SPLINE
SPL {X  -160.284, Y  +717.322, Z    +0.000, E1   -73.988, E3 +103602.756}
SPL {X  -157.512, Y  +726.783, Z    +0.000, E1   -73.653, E3 +103611.470}
SPL {X  -155.383, Y  +732.911, Z    +0.000, E1   -73.297, E3 +103618.397}
SPL {X  -152.193, Y  +740.900, Z    +0.000, E1   -73.135, E3 +103624.475}
SPL {X  -148.880, Y  +748.126, Z    +0.000, E1   -72.716, E3 +103632.256}
SPL {X  -144.434, Y  +756.610, Z    +0.000, E1   -72.338, E3 +103640.106}
SPL {X  -141.532, Y  +761.573, Z    +0.000, E1   -71.800, E3 +103646.746}
SPL {X  -138.580, Y  +766.249, Z    +0.000, E1   -71.449, E3 +103651.808}
SPL {X  -134.851, Y  +771.704, Z    +0.000, E1   -71.081, E3 +103657.203}
SPL {X  -130.513, Y  +777.511, Z    +0.000, E1   -70.561, E3 +103663.386}
SPL {X  -127.002, Y  +781.850, Z    +0.000, E1   -69.819, E3 +103669.241}
SPL {X  -118.977, Y  +790.758, Z    +0.000, E1   -71.976, E3 +103665.358}
SPL {X   -54.135, Y  +832.054, Z    +0.000, E1   -56.519, E3 +103841.284}
ENDSPLINE

SPLINE
SPL {X  -119.915, Y  +789.781, Z    +0.000, E1   -62.637, E3 +104008.899}
SPL {X  -140.675, Y  +762.967, Z    +0.000, E1   -56.489, E3 +104009.241}
SPL {X  -155.138, Y  +733.569, Z    +0.000, E1   -46.550, E3 +104011.546}
SPL {X  -162.699, Y  +706.626, Z    +0.000, E1   -30.890, E3 +104010.587}
SPL {X  -165.420, Y  +684.230, Z    +0.000, E1   -11.665, E3 +104010.338}
SPL {X  -165.650, Y  +673.379, Z    +0.000, E1    +0.036, E3 +104008.998}
SPL {X  -165.650, Y  +670.223, Z    +0.000, E1    +7.575, E3 +104008.439}
SPL {X  -165.650, Y  +666.568, Z    +0.000, E1   +16.799, E3 +104008.416}
SPL {X  -165.650, Y  +661.246, Z    +0.000, E1   +30.569, E3 +104008.196}
SPL {X  -165.650, Y  +652.403, Z    +0.000, E1   +48.665, E3 +104007.834}
SPL {X  -165.650, Y  +637.100, Z    +0.000, E1   +69.106, E3 +104004.174}
SPL {X  -165.650, Y  +616.344, Z    +0.000, E1   +74.941, E3 +104007.424}
SPL {X  -165.650, Y  +575.817, Z    +0.000, E1   +77.800, E3 +104016.353}
SPL {X  -161.405, Y  +341.238, Z    +0.000, E1   +76.606, E3 +104107.653}
SPL {X  -146.302, Y  +300.811, Z    +0.000, E1   +78.008, E3 +104108.770}
ENDSPLINE

SPLINE
SPL {X  -147.825, Y  +303.750, Z    +0.000, E1   +76.548, E3 +104123.202}
SPL {X  -148.167, Y  +304.430, Z    +0.000, E1   +75.276, E3 +104135.295}
ENDSPLINE

SPLINE
SPL {X  -146.983, Y  +302.107, Z    +0.000, E1   +74.473, E3 +104143.775}
SPL {X  -146.624, Y  +301.420, Z    +0.000, E1   +73.294, E3 +104154.259}
SPL {X  -144.830, Y  +298.101, Z    +0.000, E1   +72.333, E3 +104163.783}
SPL {X  -140.483, Y  +290.724, Z    +0.000, E1   +71.922, E3 +104170.940}
SPL {X  -135.200, Y  +282.788, Z    +0.000, E1   +71.482, E3 +104178.285}
SPL {X  -130.835, Y  +276.902, Z    +0.000, E1   +70.642, E3 +104186.187}
SPL {X  -127.149, Y  +272.325, Z    +0.000, E1   +70.073, E3 +104191.439}
SPL {X  -123.924, Y  +268.578, Z    +0.000, E1   +70.633, E3 +104191.255}
SPL {X  -115.163, Y  +259.431, Z    +0.000, E1   +74.058, E3 +104182.365}
SPL {X   -55.479, Y  +222.417, Z    +0.000, E1   +56.403, E3 +104368.218}
ENDSPLINE

SPLINE
SPL {X  -130.757, Y  +276.802, Z    +0.000, E1   +58.343, E3 +104524.155}
SPL {X  -154.788, Y  +319.502, Z    +0.000, E1   +45.389, E3 +104528.353}
SPL {X  -161.887, Y  +343.393, Z    +0.000, E1   +32.461, E3 +104528.809}
SPL {X  -164.949, Y  +363.277, Z    +0.000, E1   +17.059, E3 +104528.084}
SPL {X  -165.591, Y  +374.070, Z    +0.000, E1    +6.781, E3 +104527.747}
SPL {X  -165.650, Y  +380.752, Z    +0.000, E1    -0.182, E3 +104526.743}
SPL {X  -165.650, Y  +385.053, Z    +0.000, E1   -10.073, E3 +104526.210}
SPL {X  -165.650, Y  +388.847, Z    +0.000, E1   -19.524, E3 +104526.175}
SPL {X  -165.650, Y  +394.451, Z    +0.000, E1   -33.170, E3 +104525.588}
SPL {X  -165.650, Y  +401.692, Z    +0.000, E1   -47.300, E3 +104525.570}
SPL {X  -165.650, Y  +412.079, Z    +0.000, E1   -62.360, E3 +104523.412}
SPL {X  -165.650, Y  +422.274, Z    +0.000, E1   -68.953, E3 +104523.898}
SPL {X  -165.650, Y  +460.635, Z    +0.000, E1   -76.744, E3 +104529.469}
SPL {X  -165.650, Y  +476.745, Z    +0.000, E1   -77.150, E3 +104534.021}
SPL {X  -160.882, Y  +714.957, Z    +0.000, E1   -77.470, E3 +104615.822}
ENDSPLINE

SPLINE
SPL {X  -163.522, Y  +701.969, Z    +0.000, E1   -74.236, E3 +104645.477}
ENDSPLINE

SPLINE
SPL {X  -160.284, Y  +717.322, Z    +0.000, E1   -73.988, E3 +104656.810}
SPL {X  -157.512, Y  +726.783, Z    +0.000, E1   -73.653, E3 +104665.524}
SPL {X  -155.383, Y  +732.911, Z    +0.000, E1   -73.297, E3 +104672.451}
SPL {X  -152.193, Y  +740.900, Z    +0.000, E1   -73.135, E3 +104678.529}
SPL {X  -148.880, Y  +748.126, Z    +0.000, E1   -72.716, E3 +104686.310}
SPL {X  -144.434, Y  +756.610, Z    +0.000, E1   -72.338, E3 +104694.160}
SPL {X  -141.532, Y  +761.573, Z    +0.000, E1   -71.800, E3 +104700.800}
SPL {X  -138.580, Y  +766.249, Z    +0.000, E1   -71.449, E3 +104705.862}
SPL {X  -134.851, Y  +771.704, Z    +0.000, E1   -71.081, E3 +104711.257}
SPL {X  -130.513, Y  +777.511, Z    +0.000, E1   -70.561, E3 +104717.440}
SPL {X  -127.002, Y  +781.850, Z    +0.000, E1   -69.819, E3 +104723.295}
SPL {X  -118.977, Y  +790.758, Z    +0.000, E1   -71.976, E3 +104719.412}
SPL {X   -54.135, Y  +832.054, Z    +0.000, E1   -56.519, E3 +104895.338}
ENDSPLINE

SPLINE
SPL {X  -119.915, Y  +789.781, Z    +0.000, E1   -62.637, E3 +105062.953}
SPL {X  -140.675, Y  +762.967, Z    +0.000, E1   -56.489, E3 +105063.295}
SPL {X  -155.138, Y  +733.569, Z    +0.000, E1   -46.550, E3 +105065.600}
SPL {X  -162.699, Y  +706.626, Z    +0.000, E1   -30.890, E3 +105064.641}
SPL {X  -165.420, Y  +684.230, Z    +0.000, E1   -11.665, E3 +105064.392}
SPL {X  -165.650, Y  +673.379, Z    +0.000, E1    +0.036, E3 +105063.052}
SPL {X  -165.650, Y  +670.223, Z    +0.000, E1    +7.575, E3 +105062.493}
SPL {X  -165.650, Y  +666.568, Z    +0.000, E1   +16.799, E3 +105062.470}
SPL {X  -165.650, Y  +661.246, Z    +0.000, E1   +30.569, E3 +105062.250}
SPL {X  -165.650, Y  +652.403, Z    +0.000, E1   +48.665, E3 +105061.888}
SPL {X  -165.650, Y  +637.100, Z    +0.000, E1   +69.106, E3 +105058.228}
SPL {X  -165.650, Y  +616.344, Z    +0.000, E1   +74.941, E3 +105061.478}
SPL {X  -165.650, Y  +575.817, Z    +0.000, E1   +77.800, E3 +105070.407}
SPL {X  -162.613, Y  +346.923, Z    +0.000, E1   +78.263, E3 +105142.080}
SPL {X  -161.207, Y  +340.393, Z    +0.000, E1   +75.705, E3 +105171.943}
SPL {X  -146.302, Y  +300.811, Z    +0.000, E1   +78.008, E3 +105162.824}
ENDSPLINE

SPLINE
SPL {X  -147.825, Y  +303.750, Z    +0.000, E1   +76.548, E3 +105177.256}
SPL {X  -148.167, Y  +304.430, Z    +0.000, E1   +75.276, E3 +105189.349}
ENDSPLINE

SPLINE
SPL {X  -146.983, Y  +302.107, Z    +0.000, E1   +74.473, E3 +105197.829}
SPL {X  -146.624, Y  +301.420, Z    +0.000, E1   +73.294, E3 +105208.313}
SPL {X  -144.830, Y  +298.101, Z    +0.000, E1   +72.333, E3 +105217.837}
SPL {X  -140.483, Y  +290.724, Z    +0.000, E1   +71.922, E3 +105224.994}
SPL {X  -136.362, Y  +284.451, Z    +0.000, E1   +71.514, E3 +105231.160}
SPL {X  -133.329, Y  +280.198, Z    +0.000, E1   +71.389, E3 +105234.245}
SPL {X  -130.835, Y  +276.902, Z    +0.000, E1   +70.642, E3 +105240.241}
SPL {X  -127.149, Y  +272.325, Z    +0.000, E1   +70.073, E3 +105245.493}
SPL {X  -123.924, Y  +268.578, Z    +0.000, E1   +70.633, E3 +105245.309}
SPL {X  -115.163, Y  +259.431, Z    +0.000, E1   +74.058, E3 +105236.419}
SPL {X   -55.479, Y  +222.417, Z    +0.000, E1   +56.403, E3 +105422.272}
ENDSPLINE

SPLINE
SPL {X  -130.757, Y  +276.802, Z    +0.000, E1   +58.343, E3 +105578.209}
SPL {X  -154.788, Y  +319.502, Z    +0.000, E1   +45.389, E3 +105582.407}
SPL {X  -161.887, Y  +343.393, Z    +0.000, E1   +32.461, E3 +105582.863}
SPL {X  -164.949, Y  +363.277, Z    +0.000, E1   +17.059, E3 +105582.138}
SPL {X  -165.638, Y  +376.493, Z    +0.000, E1    +4.395, E3 +105581.777}
SPL {X  -165.650, Y  +380.500, Z    +0.000, E1    +0.000, E3 +105580.887}
SPL {X  -165.650, Y  +381.832, Z    +0.000, E1    -2.686, E3 +105580.359}
SPL {X  -165.650, Y  +385.053, Z    +0.000, E1   -10.073, E3 +105580.264}
SPL {X  -165.650, Y  +388.847, Z    +0.000, E1   -19.524, E3 +105580.229}
SPL {X  -165.650, Y  +393.562, Z    +0.000, E1   -31.212, E3 +105579.713}
SPL {X  -165.650, Y  +400.090, Z    +0.000, E1   -44.561, E3 +105579.567}
SPL {X  -165.650, Y  +415.429, Z    +0.000, E1   -64.815, E3 +105577.626}
SPL {X  -165.650, Y  +470.008, Z    +0.000, E1   -77.011, E3 +105586.170}
SPL {X  -160.882, Y  +714.957, Z    +0.000, E1   -77.470, E3 +105669.876}
ENDSPLINE

SPLINE
SPL {X  -163.522, Y  +701.969, Z    +0.000, E1   -74.236, E3 +105699.531}
ENDSPLINE

SPLINE
SPL {X  -160.284, Y  +717.322, Z    +0.000, E1   -73.988, E3 +105710.864}
SPL {X  -156.453, Y  +729.928, Z    +0.000, E1   -73.507, E3 +105723.017}
SPL {X  -152.193, Y  +740.900, Z    +0.000, E1   -73.135, E3 +105732.583}
SPL {X  -148.880, Y  +748.126, Z    +0.000, E1   -72.716, E3 +105740.364}
SPL {X  -144.434, Y  +756.610, Z    +0.000, E1   -72.338, E3 +105748.214}
SPL {X  -141.532, Y  +761.573, Z    +0.000, E1   -71.800, E3 +105754.854}
SPL {X  -138.580, Y  +766.249, Z    +0.000, E1   -71.449, E3 +105759.916}
SPL {X  -134.851, Y  +771.704, Z    +0.000, E1   -71.081, E3 +105765.311}
SPL {X  -131.668, Y  +776.015, Z    +0.000, E1   -70.566, E3 +105770.585}
SPL {X  -128.114, Y  +780.508, Z    +0.000, E1   -70.155, E3 +105775.180}
SPL {X  -123.825, Y  +785.533, Z    +0.000, E1   -70.642, E3 +105775.928}
SPL {X  -111.068, Y  +798.397, Z    +0.000, E1   -72.944, E3 +105773.373}
SPL {X   -54.135, Y  +832.054, Z    +0.000, E1   -56.519, E3 +105949.392}
ENDSPLINE

SPLINE
SPL {X  -119.915, Y  +789.781, Z    +0.000, E1   -62.637, E3 +106117.007}
SPL {X  -140.675, Y  +762.967, Z    +0.000, E1   -56.489, E3 +106117.349}
SPL {X  -155.138, Y  +733.569, Z    +0.000, E1   -46.550, E3 +106119.654}
SPL {X  -161.585, Y  +711.971, Z    +0.000, E1   -34.503, E3 +106118.704}
SPL {X  -164.796, Y  +692.295, Z    +0.000, E1   -19.289, E3 +106118.738}
SPL {X  -165.632, Y  +677.938, Z    +0.000, E1    -5.073, E3 +106118.109}
SPL {X  -165.650, Y  +673.500, Z    +0.000, E1    +0.000, E3 +106117.144}
SPL {X  -165.650, Y  +671.349, Z    +0.000, E1    +4.619, E3 +106116.648}
SPL {X  -165.650, Y  +666.568, Z    +0.000, E1   +16.799, E3 +106116.524}
SPL {X  -165.650, Y  +661.246, Z    +0.000, E1   +30.569, E3 +106116.304}
SPL {X  -165.650, Y  +655.398, Z    +0.000, E1   +43.871, E3 +106115.752}
SPL {X  -165.650, Y  +646.168, Z    +0.000, E1   +58.442, E3 +106114.846}
SPL {X  -165.650, Y  +629.125, Z    +0.000, E1   +72.389, E3 +106113.143}
SPL {X  -165.650, Y  +575.817, Z    +0.000, E1   +77.800, E3 +106124.461}
SPL {X  -161.405, Y  +341.238, Z    +0.000, E1   +76.606, E3 +106215.761}
SPL {X  -146.302, Y  +300.811, Z    +0.000, E1   +78.008, E3 +106216.878}
ENDSPLINE

SPLINE
SPL {X  -147.825, Y  +303.750, Z    +0.000, E1   +76.548, E3 +106231.310}
SPL {X  -148.167, Y  +304.430, Z    +0.000, E1   +75.276, E3 +106243.403}
ENDSPLINE

SPLINE
SPL {X  -146.983, Y  +302.107, Z    +0.000, E1   +74.473, E3 +106251.883}
SPL {X  -146.624, Y  +301.420, Z    +0.000, E1   +73.294, E3 +106262.367}
SPL {X  -144.830, Y  +298.101, Z    +0.000, E1   +72.333, E3 +106271.891}
SPL {X  -140.483, Y  +290.724, Z    +0.000, E1   +71.922, E3 +106279.048}
SPL {X  -136.362, Y  +284.451, Z    +0.000, E1   +71.514, E3 +106285.214}
SPL {X  -132.604, Y  +279.221, Z    +0.000, E1   +70.988, E3 +106291.243}
SPL {X  -129.663, Y  +275.410, Z    +0.000, E1   +70.632, E3 +106295.167}
SPL {X  -127.149, Y  +272.325, Z    +0.000, E1   +70.073, E3 +106299.547}
SPL {X  -123.924, Y  +268.578, Z    +0.000, E1   +70.633, E3 +106299.363}
SPL {X  -115.163, Y  +259.431, Z    +0.000, E1   +74.058, E3 +106290.473}
SPL {X   -55.479, Y  +222.417, Z    +0.000, E1   +56.403, E3 +106476.326}
ENDSPLINE

SPLINE
SPL {X  -130.757, Y  +276.802, Z    +0.000, E1   +58.343, E3 +106632.263}
SPL {X  -154.788, Y  +319.502, Z    +0.000, E1   +45.389, E3 +106636.461}
SPL {X  -161.887, Y  +343.393, Z    +0.000, E1   +32.461, E3 +106636.917}
SPL {X  -164.949, Y  +363.277, Z    +0.000, E1   +17.059, E3 +106636.192}
SPL {X  -165.638, Y  +376.493, Z    +0.000, E1    +4.395, E3 +106635.831}
SPL {X  -165.650, Y  +380.500, Z    +0.000, E1    +0.000, E3 +106634.941}
SPL {X  -165.650, Y  +381.832, Z    +0.000, E1    -2.686, E3 +106634.413}
SPL {X  -165.650, Y  +385.053, Z    +0.000, E1   -10.073, E3 +106634.318}
SPL {X  -165.650, Y  +388.847, Z    +0.000, E1   -19.524, E3 +106634.283}
SPL {X  -165.650, Y  +393.562, Z    +0.000, E1   -31.212, E3 +106633.767}
SPL {X  -165.650, Y  +400.090, Z    +0.000, E1   -44.561, E3 +106633.621}
SPL {X  -165.650, Y  +415.429, Z    +0.000, E1   -64.815, E3 +106631.680}
SPL {X  -165.650, Y  +470.008, Z    +0.000, E1   -77.011, E3 +106640.224}
SPL {X  -161.095, Y  +714.078, Z    +0.000, E1   -78.221, E3 +106715.759}
ENDSPLINE

SPLINE
SPL {X  -163.418, Y  +702.603, Z    +0.000, E1   -74.313, E3 +106753.155}
ENDSPLINE

SPLINE
SPL {X  -160.284, Y  +717.322, Z    +0.000, E1   -73.988, E3 +106764.918}
SPL {X  -156.453, Y  +729.928, Z    +0.000, E1   -73.507, E3 +106777.071}
SPL {X  -152.193, Y  +740.900, Z    +0.000, E1   -73.135, E3 +106786.637}
SPL {X  -148.880, Y  +748.126, Z    +0.000, E1   -72.716, E3 +106794.418}
SPL {X  -145.823, Y  +754.085, Z    +0.000, E1   -72.288, E3 +106801.190}
SPL {X  -141.906, Y  +760.955, Z    +0.000, E1   -72.057, E3 +106806.880}
SPL {X  -138.580, Y  +766.249, Z    +0.000, E1   -71.449, E3 +106813.970}
SPL {X  -134.851, Y  +771.704, Z    +0.000, E1   -71.081, E3 +106819.365}
SPL {X  -130.513, Y  +777.511, Z    +0.000, E1   -70.561, E3 +106825.548}
SPL {X  -127.002, Y  +781.850, Z    +0.000, E1   -69.819, E3 +106831.403}
SPL {X  -118.977, Y  +790.758, Z    +0.000, E1   -71.976, E3 +106827.520}
SPL {X   -54.368, Y  +831.974, Z    +0.000, E1   -57.152, E3 +106979.309}
ENDSPLINE

SPLINE
SPL {X  -111.514, Y  +797.993, Z    +0.000, E1   -63.064, E3 +107165.440}
SPL {X  -140.675, Y  +762.967, Z    +0.000, E1   -56.489, E3 +107171.403}
SPL {X  -155.138, Y  +733.569, Z    +0.000, E1   -46.550, E3 +107173.708}
SPL {X  -161.585, Y  +711.971, Z    +0.000, E1   -34.503, E3 +107172.758}
SPL {X  -164.796, Y  +692.295, Z    +0.000, E1   -19.289, E3 +107172.792}
SPL {X  -165.632, Y  +677.938, Z    +0.000, E1    -5.073, E3 +107172.163}
SPL {X  -165.650, Y  +673.500, Z    +0.000, E1    +0.000, E3 +107171.198}
SPL {X  -165.650, Y  +671.349, Z    +0.000, E1    +4.619, E3 +107170.702}
SPL {X  -165.650, Y  +666.568, Z    +0.000, E1   +16.799, E3 +107170.578}
SPL {X  -165.650, Y  +661.246, Z    +0.000, E1   +30.569, E3 +107170.358}
SPL {X  -165.650, Y  +655.398, Z    +0.000, E1   +43.871, E3 +107169.806}
SPL {X  -165.650, Y  +648.742, Z    +0.000, E1   +53.940, E3 +107170.229}
SPL {X  -165.650, Y  +637.100, Z    +0.000, E1   +69.106, E3 +107166.336}
SPL {X  -165.650, Y  +616.344, Z    +0.000, E1   +74.941, E3 +107169.586}
SPL {X  -165.650, Y  +575.817, Z    +0.000, E1   +77.800, E3 +107178.515}
SPL {X  -162.613, Y  +346.923, Z    +0.000, E1   +78.263, E3 +107250.188}
SPL {X  -161.207, Y  +340.393, Z    +0.000, E1   +75.705, E3 +107280.051}
SPL {X  -146.302, Y  +300.811, Z    +0.000, E1   +78.008, E3 +107270.932}
ENDSPLINE

SPLINE
SPL {X  -147.825, Y  +303.750, Z    +0.000, E1   +76.548, E3 +107285.364}
SPL {X  -148.167, Y  +304.430, Z    +0.000, E1   +75.276, E3 +107297.457}
ENDSPLINE

SPLINE
SPL {X  -146.983, Y  +302.107, Z    +0.000, E1   +74.473, E3 +107305.937}
SPL {X  -146.624, Y  +301.420, Z    +0.000, E1   +73.294, E3 +107316.421}
SPL {X  -144.830, Y  +298.101, Z    +0.000, E1   +72.333, E3 +107325.945}
SPL {X  -140.483, Y  +290.724, Z    +0.000, E1   +71.922, E3 +107333.102}
SPL {X  -136.362, Y  +284.451, Z    +0.000, E1   +71.514, E3 +107339.268}
SPL {X  -133.329, Y  +280.198, Z    +0.000, E1   +71.389, E3 +107342.353}
SPL {X  -130.835, Y  +276.902, Z    +0.000, E1   +70.642, E3 +107348.349}
SPL {X  -127.149, Y  +272.325, Z    +0.000, E1   +70.073, E3 +107353.601}
SPL {X  -123.924, Y  +268.578, Z    +0.000, E1   +70.633, E3 +107353.417}
SPL {X  -115.163, Y  +259.431, Z    +0.000, E1   +74.058, E3 +107344.527}
SPL {X   -55.479, Y  +222.417, Z    +0.000, E1   +56.403, E3 +107530.381}
ENDSPLINE

SPLINE
SPL {X  -130.757, Y  +276.802, Z    +0.000, E1   +58.343, E3 +107686.317}
SPL {X  -154.788, Y  +319.502, Z    +0.000, E1   +45.389, E3 +107690.515}
SPL {X  -161.887, Y  +343.393, Z    +0.000, E1   +32.461, E3 +107690.972}
SPL {X  -164.949, Y  +363.277, Z    +0.000, E1   +17.059, E3 +107690.246}
SPL {X  -165.638, Y  +376.493, Z    +0.000, E1    +4.395, E3 +107689.885}
SPL {X  -165.650, Y  +380.500, Z    +0.000, E1    +0.000, E3 +107688.995}
SPL {X  -165.650, Y  +381.832, Z    +0.000, E1    -2.686, E3 +107688.467}
SPL {X  -165.650, Y  +385.053, Z    +0.000, E1   -10.073, E3 +107688.373}
SPL {X  -165.650, Y  +388.847, Z    +0.000, E1   -19.524, E3 +107688.337}
SPL {X  -165.650, Y  +393.562, Z    +0.000, E1   -31.212, E3 +107687.821}
SPL {X  -165.650, Y  +400.090, Z    +0.000, E1   -44.561, E3 +107687.675}
SPL {X  -165.650, Y  +415.429, Z    +0.000, E1   -64.815, E3 +107685.734}
SPL {X  -165.650, Y  +470.008, Z    +0.000, E1   -77.011, E3 +107694.278}
SPL {X  -160.882, Y  +714.957, Z    +0.000, E1   -77.470, E3 +107777.984}
ENDSPLINE

SPLINE
SPL {X  -163.522, Y  +701.969, Z    +0.000, E1   -74.236, E3 +107807.639}
ENDSPLINE

SPLINE
SPL {X  -160.284, Y  +717.322, Z    +0.000, E1   -73.988, E3 +107818.973}
SPL {X  -156.453, Y  +729.928, Z    +0.000, E1   -73.507, E3 +107831.125}
SPL {X  -152.193, Y  +740.900, Z    +0.000, E1   -73.135, E3 +107840.691}
SPL {X  -148.880, Y  +748.126, Z    +0.000, E1   -72.716, E3 +107848.472}
SPL {X  -144.434, Y  +756.610, Z    +0.000, E1   -72.338, E3 +107856.322}
SPL {X  -141.532, Y  +761.573, Z    +0.000, E1   -71.800, E3 +107862.963}
SPL {X  -138.580, Y  +766.249, Z    +0.000, E1   -71.449, E3 +107868.024}
SPL {X  -134.851, Y  +771.704, Z    +0.000, E1   -71.081, E3 +107873.419}
SPL {X  -131.668, Y  +776.015, Z    +0.000, E1   -70.566, E3 +107878.693}
SPL {X  -128.114, Y  +780.508, Z    +0.000, E1   -70.155, E3 +107883.288}
SPL {X  -123.825, Y  +785.533, Z    +0.000, E1   -70.642, E3 +107884.036}
SPL {X  -111.068, Y  +798.397, Z    +0.000, E1   -72.944, E3 +107881.481}
SPL {X   -54.135, Y  +832.054, Z    +0.000, E1   -56.519, E3 +108057.500}
ENDSPLINE

SPLINE
SPL {X  -119.915, Y  +789.781, Z    +0.000, E1   -62.637, E3 +108225.115}
SPL {X  -140.675, Y  +762.967, Z    +0.000, E1   -56.489, E3 +108225.457}
SPL {X  -155.138, Y  +733.569, Z    +0.000, E1   -46.550, E3 +108227.762}
SPL {X  -161.585, Y  +711.971, Z    +0.000, E1   -34.503, E3 +108226.812}
SPL {X  -164.796, Y  +692.295, Z    +0.000, E1   -19.289, E3 +108226.847}
SPL {X  -165.632, Y  +677.938, Z    +0.000, E1    -5.073, E3 +108226.218}
SPL {X  -165.650, Y  +673.500, Z    +0.000, E1    +0.000, E3 +108225.252}
SPL {X  -165.650, Y  +671.349, Z    +0.000, E1    +4.619, E3 +108224.756}
SPL {X  -165.650, Y  +666.568, Z    +0.000, E1   +16.799, E3 +108224.632}
SPL {X  -165.650, Y  +661.246, Z    +0.000, E1   +30.569, E3 +108224.412}
SPL {X  -165.650, Y  +652.403, Z    +0.000, E1   +48.665, E3 +108224.050}
SPL {X  -165.650, Y  +637.100, Z    +0.000, E1   +69.106, E3 +108220.390}
SPL {X  -165.650, Y  +616.344, Z    +0.000, E1   +74.941, E3 +108223.640}
SPL {X  -165.650, Y  +575.817, Z    +0.000, E1   +77.800, E3 +108232.569}
SPL {X  -161.405, Y  +341.238, Z    +0.000, E1   +76.606, E3 +108323.869}
SPL {X  -146.302, Y  +300.811, Z    +0.000, E1   +78.008, E3 +108324.986}
ENDSPLINE

SPLINE
SPL {X  -147.825, Y  +303.750, Z    +0.000, E1   +76.548, E3 +108339.418}
SPL {X  -148.167, Y  +304.430, Z    +0.000, E1   +75.276, E3 +108351.511}
ENDSPLINE

SPLINE
SPL {X  -146.983, Y  +302.107, Z    +0.000, E1   +74.473, E3 +108359.992}
ENDSPLINE

SPLINE
SPL {X  -147.081, Y  +302.295, Z    +0.000, E1   +73.151, E3 +108371.252}
SPL {X  -152.732, Y  +314.368, Z    +0.000, E1   +69.769, E3 +108390.935}
ENDSPLINE

SPLINE
SPL {X  -149.246, Y  +306.628, Z    +0.000, E1   +69.029, E3 +108401.808}
SPL {X  -144.614, Y  +297.712, Z    +0.000, E1   +68.717, E3 +108410.161}
SPL {X  -141.011, Y  +291.576, Z    +0.000, E1   +68.040, E3 +108418.639}
SPL {X  -137.649, Y  +286.345, Z    +0.000, E1   +67.498, E3 +108425.333}
SPL {X  -134.450, Y  +281.737, Z    +0.000, E1   +67.268, E3 +108429.723}
SPL {X  -131.812, Y  +278.173, Z    +0.000, E1   +66.669, E3 +108435.071}
SPL {X  -128.148, Y  +273.533, Z    +0.000, E1   +67.328, E3 +108435.430}
SPL {X  -116.216, Y  +260.459, Z    +0.000, E1   +70.200, E3 +108431.736}
SPL {X   -66.125, Y  +226.621, Z    +0.000, E1   +55.862, E3 +108594.634}
ENDSPLINE

SPLINE
SPL {X  -111.531, Y  +256.023, Z    +0.000, E1   +58.853, E3 +108737.516}
SPL {X  -139.240, Y  +288.767, Z    +0.000, E1   +52.898, E3 +108747.689}
SPL {X  -156.827, Y  +325.161, Z    +0.000, E1   +39.042, E3 +108746.059}
SPL {X  -162.324, Y  +345.471, Z    +0.000, E1   +27.849, E3 +108746.527}
SPL {X  -165.055, Y  +364.477, Z    +0.000, E1   +14.326, E3 +108746.965}
SPL {X  -165.646, Y  +377.353, Z    +0.000, E1    +3.112, E3 +108745.922}
SPL {X  -165.650, Y  +380.500, Z    +0.000, E1    -0.000, E3 +108745.048}
SPL {X  -165.650, Y  +381.828, Z    +0.000, E1    -2.219, E3 +108744.501}
SPL {X  -165.650, Y  +385.044, Z    +0.000, E1    -8.496, E3 +108744.300}
SPL {X  -165.650, Y  +388.717, Z    +0.000, E1   -16.400, E3 +108744.156}
SPL {X  -165.650, Y  +394.613, Z    +0.000, E1   -29.184, E3 +108743.625}
SPL {X  -165.650, Y  +402.836, Z    +0.000, E1   -44.797, E3 +108743.027}
SPL {X  -165.650, Y  +416.111, Z    +0.000, E1   -60.729, E3 +108742.094}
SPL {X  -165.650, Y  +471.994, Z    +0.000, E1   -75.670, E3 +108750.147}
SPL {X  -164.204, Y  +697.342, Z    +0.000, E1   -76.015, E3 +108838.170}
ENDSPLINE

SPLINE
SPL {X  -165.650, Y  +656.030, Z    +0.000, E1   -71.686, E3 +108859.610}
ENDSPLINE

SPLINE
SPL {X  -165.610, Y  +679.119, Z    +0.000, E1   -71.889, E3 +108873.233}
SPL {X  -164.561, Y  +694.465, Z    +0.000, E1   -71.736, E3 +108884.866}
SPL {X  -162.089, Y  +709.665, Z    +0.000, E1   -71.739, E3 +108895.067}
SPL {X  -159.776, Y  +719.221, Z    +0.000, E1   -71.038, E3 +108907.889}
SPL {X  -155.811, Y  +731.738, Z    +0.000, E1   -70.890, E3 +108917.577}
SPL {X  -152.643, Y  +739.844, Z    +0.000, E1   -70.463, E3 +108926.436}
SPL {X  -149.782, Y  +746.247, Z    +0.000, E1   -70.149, E3 +108933.126}
SPL {X  -146.450, Y  +752.910, Z    +0.000, E1   -69.680, E3 +108941.004}
SPL {X  -143.017, Y  +759.082, Z    +0.000, E1   -69.156, E3 +108948.615}
SPL {X  -140.057, Y  +763.953, Z    +0.000, E1   -68.829, E3 +108953.855}
SPL {X  -136.535, Y  +769.298, Z    +0.000, E1   -68.442, E3 +108959.716}
SPL {X  -133.553, Y  +773.498, Z    +0.000, E1   -67.773, E3 +108965.881}
SPL {X  -129.830, Y  +778.379, Z    +0.000, E1   -67.491, E3 +108970.507}
SPL {X  -116.788, Y  +792.975, Z    +0.000, E1   -71.297, E3 +108963.891}
SPL {X   -64.927, Y  +827.895, Z    +0.000, E1   -57.691, E3 +109089.494}
ENDSPLINE

SPLINE
SPL {X  -111.648, Y  +797.871, Z    +0.000, E1   -60.847, E3 +109286.477}
SPL {X  -149.288, Y  +747.285, Z    +0.000, E1   -46.770, E3 +109282.468}
SPL {X  -159.627, Y  +719.761, Z    +0.000, E1   -35.247, E3 +109287.533}
SPL {X  -164.185, Y  +697.485, Z    +0.000, E1   -20.950, E3 +109287.852}
SPL {X  -165.594, Y  +679.817, Z    +0.000, E1    -6.204, E3 +109286.628}
SPL {X  -165.650, Y  +673.522, Z    +0.000, E1    -0.038, E3 +109285.597}
SPL {X  -165.650, Y  +671.354, Z    +0.000, E1    +3.728, E3 +109285.085}
SPL {X  -165.650, Y  +666.485, Z    +0.000, E1   +14.169, E3 +109284.812}
SPL {X  -165.650, Y  +661.236, Z    +0.000, E1   +26.072, E3 +109284.501}
SPL {X  -165.650, Y  +653.063, Z    +0.000, E1   +42.395, E3 +109283.905}
SPL {X  -165.650, Y  +640.535, Z    +0.000, E1   +60.776, E3 +109281.390}
SPL {X  -165.650, Y  +618.963, Z    +0.000, E1   +72.815, E3 +109281.369}
SPL {X  -165.650, Y  +582.897, Z    +0.000, E1   +76.147, E3 +109290.030}
SPL {X  -165.650, Y  +558.388, Z    +0.000, E1   +76.294, E3 +109298.342}
SPL {X  -165.650, Y  +391.690, Z    +0.000, E1   +75.504, E3 +109368.108}
ENDSPLINE

SPLINE
SPL {X  -165.650, Y  +396.283, Z    +0.000, E1   +72.775, E3 +109391.413}
SPL {X  -165.650, Y  +407.500, Z    +0.000, E1   +70.919, E3 +109402.397}
ENDSPLINE

SPLINE
SPL {X  -165.650, Y  +384.687, Z    +0.000, E1   +71.028, E3 +109417.643}
SPL {X  -164.996, Y  +363.797, Z    +0.000, E1   +70.987, E3 +109432.618}
SPL {X  -162.841, Y  +348.123, Z    +0.000, E1   +70.683, E3 +109446.546}
SPL {X  -162.352, Y  +345.609, Z    +0.000, E1   +69.290, E3 +109460.499}
SPL {X  -157.663, Y  +327.685, Z    +0.000, E1   +69.808, E3 +109469.359}
SPL {X  -152.892, Y  +314.750, Z    +0.000, E1   +69.675, E3 +109479.575}
SPL {X  -149.246, Y  +306.628, Z    +0.000, E1   +69.029, E3 +109490.043}
SPL {X  -144.614, Y  +297.712, Z    +0.000, E1   +68.717, E3 +109498.396}
SPL {X  -141.011, Y  +291.576, Z    +0.000, E1   +68.040, E3 +109506.875}
SPL {X  -137.649, Y  +286.345, Z    +0.000, E1   +67.498, E3 +109513.568}
SPL {X  -134.450, Y  +281.737, Z    +0.000, E1   +67.268, E3 +109517.958}
SPL {X  -131.812, Y  +278.173, Z    +0.000, E1   +66.669, E3 +109523.307}
SPL {X  -128.148, Y  +273.533, Z    +0.000, E1   +67.328, E3 +109523.665}
SPL {X  -116.216, Y  +260.459, Z    +0.000, E1   +70.200, E3 +109519.972}
SPL {X   -66.125, Y  +226.621, Z    +0.000, E1   +55.862, E3 +109682.870}
ENDSPLINE

SPLINE
SPL {X  -111.531, Y  +256.023, Z    +0.000, E1   +58.853, E3 +109825.752}
SPL {X  -139.240, Y  +288.767, Z    +0.000, E1   +52.898, E3 +109835.925}
SPL {X  -156.827, Y  +325.161, Z    +0.000, E1   +39.042, E3 +109834.294}
SPL {X  -162.324, Y  +345.471, Z    +0.000, E1   +27.849, E3 +109834.762}
SPL {X  -165.055, Y  +364.477, Z    +0.000, E1   +14.326, E3 +109835.201}
SPL {X  -165.646, Y  +377.353, Z    +0.000, E1    +3.112, E3 +109834.158}
SPL {X  -165.650, Y  +380.500, Z    +0.000, E1    -0.000, E3 +109833.284}
SPL {X  -165.650, Y  +381.828, Z    +0.000, E1    -2.219, E3 +109832.736}
SPL {X  -165.650, Y  +385.044, Z    +0.000, E1    -8.496, E3 +109832.535}
SPL {X  -165.650, Y  +388.717, Z    +0.000, E1   -16.400, E3 +109832.391}
SPL {X  -165.650, Y  +394.613, Z    +0.000, E1   -29.184, E3 +109831.860}
SPL {X  -165.650, Y  +402.836, Z    +0.000, E1   -44.797, E3 +109831.263}
SPL {X  -165.650, Y  +416.111, Z    +0.000, E1   -60.729, E3 +109830.329}
SPL {X  -165.650, Y  +471.994, Z    +0.000, E1   -75.670, E3 +109838.383}
SPL {X  -164.204, Y  +697.342, Z    +0.000, E1   -76.015, E3 +109926.405}
ENDSPLINE

SPLINE
SPL {X  -165.650, Y  +656.030, Z    +0.000, E1   -71.686, E3 +109947.845}
ENDSPLINE

SPLINE
SPL {X  -165.610, Y  +679.119, Z    +0.000, E1   -71.889, E3 +109961.468}
SPL {X  -164.561, Y  +694.465, Z    +0.000, E1   -71.736, E3 +109973.101}
SPL {X  -162.089, Y  +709.665, Z    +0.000, E1   -71.739, E3 +109983.302}
SPL {X  -159.776, Y  +719.221, Z    +0.000, E1   -71.038, E3 +109996.124}
SPL {X  -155.811, Y  +731.738, Z    +0.000, E1   -70.890, E3 +110005.812}
SPL {X  -152.643, Y  +739.844, Z    +0.000, E1   -70.463, E3 +110014.672}
SPL {X  -149.782, Y  +746.247, Z    +0.000, E1   -70.149, E3 +110021.361}
SPL {X  -146.450, Y  +752.910, Z    +0.000, E1   -69.680, E3 +110029.239}
SPL {X  -143.017, Y  +759.082, Z    +0.000, E1   -69.156, E3 +110036.851}
SPL {X  -140.057, Y  +763.953, Z    +0.000, E1   -68.829, E3 +110042.090}
SPL {X  -136.535, Y  +769.298, Z    +0.000, E1   -68.442, E3 +110047.952}
SPL {X  -133.553, Y  +773.498, Z    +0.000, E1   -67.773, E3 +110054.117}
SPL {X  -129.830, Y  +778.379, Z    +0.000, E1   -67.491, E3 +110058.742}
SPL {X  -116.788, Y  +792.975, Z    +0.000, E1   -71.297, E3 +110052.127}
SPL {X   -64.927, Y  +827.895, Z    +0.000, E1   -57.691, E3 +110177.730}
ENDSPLINE

SPLINE
SPL {X  -111.648, Y  +797.871, Z    +0.000, E1   -60.847, E3 +110374.712}
SPL {X  -149.288, Y  +747.285, Z    +0.000, E1   -46.770, E3 +110370.703}
SPL {X  -159.627, Y  +719.761, Z    +0.000, E1   -35.247, E3 +110375.768}
SPL {X  -164.185, Y  +697.485, Z    +0.000, E1   -20.950, E3 +110376.087}
SPL {X  -165.594, Y  +679.817, Z    +0.000, E1    -6.204, E3 +110374.863}
SPL {X  -165.650, Y  +673.522, Z    +0.000, E1    -0.038, E3 +110373.832}
SPL {X  -165.650, Y  +671.354, Z    +0.000, E1    +3.728, E3 +110373.320}
SPL {X  -165.650, Y  +666.485, Z    +0.000, E1   +14.169, E3 +110373.047}
SPL {X  -165.650, Y  +661.236, Z    +0.000, E1   +26.072, E3 +110372.736}
SPL {X  -165.650, Y  +653.063, Z    +0.000, E1   +42.395, E3 +110372.140}
SPL {X  -165.650, Y  +640.535, Z    +0.000, E1   +60.776, E3 +110369.625}
SPL {X  -165.650, Y  +618.963, Z    +0.000, E1   +72.815, E3 +110369.604}
SPL {X  -165.650, Y  +582.897, Z    +0.000, E1   +76.147, E3 +110378.265}
SPL {X  -165.650, Y  +558.388, Z    +0.000, E1   +76.294, E3 +110386.577}
SPL {X  -165.650, Y  +391.690, Z    +0.000, E1   +75.504, E3 +110456.344}
ENDSPLINE

SPLINE
SPL {X  -165.650, Y  +396.283, Z    +0.000, E1   +72.775, E3 +110479.649}
SPL {X  -165.650, Y  +407.500, Z    +0.000, E1   +70.919, E3 +110490.632}
ENDSPLINE

SPLINE
SPL {X  -165.650, Y  +390.855, Z    +0.000, E1   +71.004, E3 +110501.560}
SPL {X  -165.534, Y  +372.295, Z    +0.000, E1   +71.066, E3 +110514.110}
SPL {X  -164.039, Y  +355.451, Z    +0.000, E1   +70.703, E3 +110529.509}
SPL {X  -161.297, Y  +340.777, Z    +0.000, E1   +70.794, E3 +110538.801}
ENDSPLINE

SPLINE
SPL {X  -162.352, Y  +345.609, Z    +0.000, E1   +69.290, E3 +110548.734}
ENDSPLINE

SPLINE
SPL {X  -159.253, Y  +332.909, Z    +0.000, E1   +69.652, E3 +110555.081}
SPL {X  -155.267, Y  +320.775, Z    +0.000, E1   +69.854, E3 +110562.174}
SPL {X  -151.256, Y  +310.961, Z    +0.000, E1   +69.467, E3 +110572.049}
SPL {X  -148.628, Y  +305.359, Z    +0.000, E1   +68.848, E3 +110580.327}
SPL {X  -145.495, Y  +299.310, Z    +0.000, E1   +68.659, E3 +110585.887}
SPL {X  -142.111, Y  +293.387, Z    +0.000, E1   +68.421, E3 +110591.528}
SPL {X  -138.525, Y  +287.667, Z    +0.000, E1   +67.662, E3 +110600.088}
SPL {X  -134.450, Y  +281.737, Z    +0.000, E1   +67.268, E3 +110606.193}
SPL {X  -131.812, Y  +278.173, Z    +0.000, E1   +66.669, E3 +110611.542}
SPL {X  -128.148, Y  +273.533, Z    +0.000, E1   +67.328, E3 +110611.900}
SPL {X  -116.216, Y  +260.459, Z    +0.000, E1   +70.200, E3 +110608.207}
SPL {X   -66.125, Y  +226.621, Z    +0.000, E1   +55.862, E3 +110771.105}
ENDSPLINE

SPLINE
SPL {X  -111.531, Y  +256.023, Z    +0.000, E1   +58.853, E3 +110913.987}
SPL {X  -139.240, Y  +288.767, Z    +0.000, E1   +52.898, E3 +110924.160}
SPL {X  -156.827, Y  +325.161, Z    +0.000, E1   +39.042, E3 +110922.529}
SPL {X  -162.324, Y  +345.471, Z    +0.000, E1   +27.849, E3 +110922.998}
SPL {X  -165.055, Y  +364.477, Z    +0.000, E1   +14.326, E3 +110923.436}
SPL {X  -165.646, Y  +377.353, Z    +0.000, E1    +3.112, E3 +110922.393}
SPL {X  -165.650, Y  +380.500, Z    +0.000, E1    -0.000, E3 +110921.519}
SPL {X  -165.650, Y  +381.828, Z    +0.000, E1    -2.219, E3 +110920.971}
SPL {X  -165.650, Y  +385.044, Z    +0.000, E1    -8.496, E3 +110920.771}
SPL {X  -165.650, Y  +388.717, Z    +0.000, E1   -16.400, E3 +110920.627}
SPL {X  -165.650, Y  +394.613, Z    +0.000, E1   -29.184, E3 +110920.095}
SPL {X  -165.650, Y  +402.836, Z    +0.000, E1   -44.797, E3 +110919.498}
SPL {X  -165.650, Y  +416.111, Z    +0.000, E1   -60.729, E3 +110918.565}
SPL {X  -165.650, Y  +471.994, Z    +0.000, E1   -75.670, E3 +110926.618}
SPL {X  -164.204, Y  +697.342, Z    +0.000, E1   -76.015, E3 +111014.641}
ENDSPLINE

SPLINE
SPL {X  -165.650, Y  +656.030, Z    +0.000, E1   -71.686, E3 +111036.080}
ENDSPLINE

SPLINE
SPL {X  -165.610, Y  +679.119, Z    +0.000, E1   -71.889, E3 +111049.703}
SPL {X  -164.561, Y  +694.465, Z    +0.000, E1   -71.736, E3 +111061.337}
SPL {X  -162.089, Y  +709.665, Z    +0.000, E1   -71.739, E3 +111071.537}
SPL {X  -159.776, Y  +719.221, Z    +0.000, E1   -71.038, E3 +111084.360}
SPL {X  -155.811, Y  +731.738, Z    +0.000, E1   -70.890, E3 +111094.048}
SPL {X  -152.643, Y  +739.844, Z    +0.000, E1   -70.463, E3 +111102.907}
SPL {X  -149.782, Y  +746.247, Z    +0.000, E1   -70.149, E3 +111109.597}
SPL {X  -146.450, Y  +752.910, Z    +0.000, E1   -69.680, E3 +111117.475}
SPL {X  -143.017, Y  +759.082, Z    +0.000, E1   -69.156, E3 +111125.086}
SPL {X  -139.030, Y  +765.558, Z    +0.000, E1   -68.719, E3 +111132.119}
SPL {X  -135.682, Y  +770.527, Z    +0.000, E1   -68.337, E3 +111137.503}
SPL {X  -132.359, Y  +775.105, Z    +0.000, E1   -67.661, E3 +111144.044}
SPL {X  -128.720, Y  +779.765, Z    +0.000, E1   -67.454, E3 +111148.025}
SPL {X  -116.788, Y  +792.975, Z    +0.000, E1   -71.297, E3 +111140.362}
SPL {X   -64.927, Y  +827.895, Z    +0.000, E1   -57.691, E3 +111265.965}
ENDSPLINE

SPLINE
SPL {X  -111.648, Y  +797.871, Z    +0.000, E1   -60.847, E3 +111462.947}
SPL {X  -149.288, Y  +747.285, Z    +0.000, E1   -46.770, E3 +111458.938}
SPL {X  -159.627, Y  +719.761, Z    +0.000, E1   -35.247, E3 +111464.003}
SPL {X  -164.185, Y  +697.485, Z    +0.000, E1   -20.950, E3 +111464.322}
SPL {X  -165.594, Y  +679.817, Z    +0.000, E1    -6.204, E3 +111463.099}
SPL {X  -165.650, Y  +673.522, Z    +0.000, E1    -0.038, E3 +111462.068}
SPL {X  -165.650, Y  +671.354, Z    +0.000, E1    +3.728, E3 +111461.555}
SPL {X  -165.650, Y  +666.485, Z    +0.000, E1   +14.169, E3 +111461.282}
SPL {X  -165.650, Y  +661.236, Z    +0.000, E1   +26.072, E3 +111460.971}
SPL {X  -165.650, Y  +653.063, Z    +0.000, E1   +42.395, E3 +111460.375}
SPL {X  -165.650, Y  +640.535, Z    +0.000, E1   +60.776, E3 +111457.860}
SPL {X  -165.650, Y  +618.963, Z    +0.000, E1   +72.815, E3 +111457.839}
SPL {X  -165.650, Y  +575.208, Z    +0.000, E1   +76.222, E3 +111469.100}
SPL {X  -165.650, Y  +394.754, Z    +0.000, E1   +73.248, E3 +111564.246}
ENDSPLINE

SPLINE
SPL {X  -165.650, Y  +407.500, Z    +0.000, E1   +70.919, E3 +111578.868}
ENDSPLINE

SPLINE
SPL {X  -165.650, Y  +390.855, Z    +0.000, E1   +71.004, E3 +111589.795}
SPL {X  -165.534, Y  +372.295, Z    +0.000, E1   +71.066, E3 +111602.346}
SPL {X  -164.039, Y  +355.451, Z    +0.000, E1   +70.703, E3 +111617.744}
SPL {X  -161.297, Y  +340.777, Z    +0.000, E1   +70.794, E3 +111627.036}
ENDSPLINE

SPLINE
SPL {X  -162.352, Y  +345.609, Z    +0.000, E1   +69.290, E3 +111636.969}
ENDSPLINE

SPLINE
SPL {X  -159.253, Y  +332.909, Z    +0.000, E1   +69.652, E3 +111643.316}
SPL {X  -155.267, Y  +320.775, Z    +0.000, E1   +69.854, E3 +111650.409}
SPL {X  -151.256, Y  +310.961, Z    +0.000, E1   +69.467, E3 +111660.284}
SPL {X  -148.628, Y  +305.359, Z    +0.000, E1   +68.848, E3 +111668.563}
SPL {X  -145.495, Y  +299.310, Z    +0.000, E1   +68.659, E3 +111674.122}
SPL {X  -142.111, Y  +293.387, Z    +0.000, E1   +68.421, E3 +111679.764}
SPL {X  -138.525, Y  +287.667, Z    +0.000, E1   +67.662, E3 +111688.323}
SPL {X  -134.450, Y  +281.737, Z    +0.000, E1   +67.268, E3 +111694.429}
SPL {X  -131.812, Y  +278.173, Z    +0.000, E1   +66.669, E3 +111699.777}
SPL {X  -128.148, Y  +273.533, Z    +0.000, E1   +67.328, E3 +111700.136}
SPL {X  -116.216, Y  +260.459, Z    +0.000, E1   +70.200, E3 +111696.442}
SPL {X   -66.125, Y  +226.621, Z    +0.000, E1   +55.862, E3 +111859.340}
ENDSPLINE

SPLINE
SPL {X  -111.531, Y  +256.023, Z    +0.000, E1   +58.853, E3 +112002.222}
SPL {X  -139.240, Y  +288.767, Z    +0.000, E1   +52.898, E3 +112012.395}
SPL {X  -156.827, Y  +325.161, Z    +0.000, E1   +39.042, E3 +112010.764}
SPL {X  -162.324, Y  +345.471, Z    +0.000, E1   +27.849, E3 +112011.233}
SPL {X  -164.696, Y  +360.744, Z    +0.000, E1   +17.229, E3 +112012.147}
SPL {X  -165.561, Y  +373.081, Z    +0.000, E1    +6.973, E3 +112010.891}
SPL {X  -165.650, Y  +380.392, Z    +0.000, E1    +0.180, E3 +112009.808}
SPL {X  -165.650, Y  +381.828, Z    +0.000, E1    -2.219, E3 +112009.206}
SPL {X  -165.650, Y  +385.044, Z    +0.000, E1    -8.496, E3 +112009.006}
SPL {X  -165.650, Y  +390.492, Z    +0.000, E1   -20.084, E3 +112008.660}
SPL {X  -165.650, Y  +400.081, Z    +0.000, E1   -39.836, E3 +112007.966}
SPL {X  -165.650, Y  +416.111, Z    +0.000, E1   -60.729, E3 +112006.800}
SPL {X  -165.650, Y  +471.994, Z    +0.000, E1   -75.670, E3 +112014.853}
SPL {X  -164.204, Y  +697.342, Z    +0.000, E1   -76.015, E3 +112102.876}
ENDSPLINE

SPLINE
SPL {X  -165.650, Y  +664.340, Z    +0.000, E1   -71.862, E3 +112128.279}
ENDSPLINE

SPLINE
SPL {X  -165.116, Y  +688.792, Z    +0.000, E1   -71.759, E3 +112145.719}
SPL {X  -162.089, Y  +709.665, Z    +0.000, E1   -71.739, E3 +112159.773}
SPL {X  -160.450, Y  +716.681, Z    +0.000, E1   -71.166, E3 +112169.576}
SPL {X  -159.124, Y  +721.538, Z    +0.000, E1   -70.872, E3 +112175.503}
SPL {X  -155.811, Y  +731.738, Z    +0.000, E1   -70.890, E3 +112182.283}
SPL {X  -152.643, Y  +739.844, Z    +0.000, E1   -70.463, E3 +112191.142}
SPL {X  -149.782, Y  +746.247, Z    +0.000, E1   -70.149, E3 +112197.832}
SPL {X  -146.450, Y  +752.910, Z    +0.000, E1   -69.680, E3 +112205.710}
SPL {X  -143.017, Y  +759.082, Z    +0.000, E1   -69.156, E3 +112213.321}
SPL {X  -140.057, Y  +763.953, Z    +0.000, E1   -68.829, E3 +112218.561}
SPL {X  -136.535, Y  +769.298, Z    +0.000, E1   -68.442, E3 +112224.422}
SPL {X  -133.553, Y  +773.498, Z    +0.000, E1   -67.773, E3 +112230.587}
SPL {X  -129.830, Y  +778.379, Z    +0.000, E1   -67.491, E3 +112235.213}
SPL {X  -116.788, Y  +792.975, Z    +0.000, E1   -71.297, E3 +112228.597}
SPL {X   -64.927, Y  +827.895, Z    +0.000, E1   -57.691, E3 +112354.200}
ENDSPLINE

SPLINE
SPL {X  -111.648, Y  +797.871, Z    +0.000, E1   -60.847, E3 +112551.183}
SPL {X  -149.288, Y  +747.285, Z    +0.000, E1   -46.770, E3 +112547.173}
SPL {X  -159.627, Y  +719.761, Z    +0.000, E1   -35.247, E3 +112552.239}
SPL {X  -164.185, Y  +697.485, Z    +0.000, E1   -20.950, E3 +112552.557}
SPL {X  -165.594, Y  +679.817, Z    +0.000, E1    -6.204, E3 +112551.334}
SPL {X  -165.650, Y  +673.522, Z    +0.000, E1    -0.038, E3 +112550.303}
SPL {X  -165.650, Y  +671.354, Z    +0.000, E1    +3.728, E3 +112549.790}
SPL {X  -165.650, Y  +666.485, Z    +0.000, E1   +14.169, E3 +112549.518}
SPL {X  -165.650, Y  +661.236, Z    +0.000, E1   +26.072, E3 +112549.207}
SPL {X  -165.650, Y  +653.063, Z    +0.000, E1   +42.395, E3 +112548.611}
SPL {X  -165.650, Y  +640.535, Z    +0.000, E1   +60.776, E3 +112546.096}
SPL {X  -165.650, Y  +618.963, Z    +0.000, E1   +72.815, E3 +112546.075}
SPL {X  -165.650, Y  +575.208, Z    +0.000, E1   +76.222, E3 +112557.335}
SPL {X  -165.650, Y  +394.754, Z    +0.000, E1   +73.248, E3 +112652.482}
ENDSPLINE

SPLINE
SPL {X  -165.650, Y  +407.500, Z    +0.000, E1   +70.919, E3 +112667.103}
ENDSPLINE

SPLINE
SPL {X  -165.650, Y  +390.855, Z    +0.000, E1   +71.004, E3 +112678.031}
SPL {X  -165.534, Y  +372.295, Z    +0.000, E1   +71.066, E3 +112690.581}
SPL {X  -164.039, Y  +355.451, Z    +0.000, E1   +70.703, E3 +112705.979}
SPL {X  -161.297, Y  +340.777, Z    +0.000, E1   +70.794, E3 +112715.272}
ENDSPLINE

SPLINE
SPL {X  -162.352, Y  +345.609, Z    +0.000, E1   +69.290, E3 +112725.205}
ENDSPLINE

SPLINE
SPL {X  -157.663, Y  +327.685, Z    +0.000, E1   +69.808, E3 +112734.065}
SPL {X  -152.892, Y  +314.750, Z    +0.000, E1   +69.675, E3 +112744.281}
SPL {X  -149.246, Y  +306.628, Z    +0.000, E1   +69.029, E3 +112754.749}
SPL {X  -145.495, Y  +299.310, Z    +0.000, E1   +68.659, E3 +112762.357}
SPL {X  -142.111, Y  +293.387, Z    +0.000, E1   +68.421, E3 +112767.999}
SPL {X  -138.525, Y  +287.667, Z    +0.000, E1   +67.662, E3 +112776.559}
SPL {X  -134.450, Y  +281.737, Z    +0.000, E1   +67.268, E3 +112782.664}
SPL {X  -131.812, Y  +278.173, Z    +0.000, E1   +66.669, E3 +112788.012}
SPL {X  -128.148, Y  +273.533, Z    +0.000, E1   +67.328, E3 +112788.371}
SPL {X  -116.216, Y  +260.459, Z    +0.000, E1   +70.200, E3 +112784.677}
SPL {X   -66.125, Y  +226.621, Z    +0.000, E1   +55.862, E3 +112947.576}
ENDSPLINE

SPLINE
SPL {X  -111.531, Y  +256.023, Z    +0.000, E1   +58.853, E3 +113090.458}
SPL {X  -139.240, Y  +288.767, Z    +0.000, E1   +52.898, E3 +113100.630}
SPL {X  -156.827, Y  +325.161, Z    +0.000, E1   +39.042, E3 +113099.000}
SPL {X  -162.324, Y  +345.471, Z    +0.000, E1   +27.849, E3 +113099.468}
SPL {X  -165.055, Y  +364.477, Z    +0.000, E1   +14.326, E3 +113099.907}
SPL {X  -165.646, Y  +377.353, Z    +0.000, E1    +3.112, E3 +113098.864}
SPL {X  -165.650, Y  +380.500, Z    +0.000, E1    -0.000, E3 +113097.989}
SPL {X  -165.650, Y  +381.828, Z    +0.000, E1    -2.219, E3 +113097.442}
SPL {X  -165.650, Y  +385.044, Z    +0.000, E1    -8.496, E3 +113097.241}
SPL {X  -165.650, Y  +390.492, Z    +0.000, E1   -20.084, E3 +113096.896}
SPL {X  -165.650, Y  +400.081, Z    +0.000, E1   -39.836, E3 +113096.201}
SPL {X  -165.650, Y  +416.111, Z    +0.000, E1   -60.729, E3 +113095.035}
SPL {X  -165.650, Y  +471.994, Z    +0.000, E1   -75.670, E3 +113103.088}
SPL {X  -164.204, Y  +697.342, Z    +0.000, E1   -76.015, E3 +113191.111}
ENDSPLINE

SPLINE
SPL {X  -165.650, Y  +664.340, Z    +0.000, E1   -71.862, E3 +113216.515}
ENDSPLINE

SPLINE
SPL {X  -165.116, Y  +688.792, Z    +0.000, E1   -71.759, E3 +113233.954}
SPL {X  -162.089, Y  +709.665, Z    +0.000, E1   -71.739, E3 +113248.008}
SPL {X  -160.450, Y  +716.681, Z    +0.000, E1   -71.166, E3 +113257.811}
SPL {X  -159.124, Y  +721.538, Z    +0.000, E1   -70.872, E3 +113263.738}
SPL {X  -155.811, Y  +731.738, Z    +0.000, E1   -70.890, E3 +113270.518}
SPL {X  -152.643, Y  +739.844, Z    +0.000, E1   -70.463, E3 +113279.377}
SPL {X  -149.782, Y  +746.247, Z    +0.000, E1   -70.149, E3 +113286.067}
SPL {X  -146.450, Y  +752.910, Z    +0.000, E1   -69.680, E3 +113293.945}
SPL {X  -143.017, Y  +759.082, Z    +0.000, E1   -69.156, E3 +113301.557}
SPL {X  -139.030, Y  +765.558, Z    +0.000, E1   -68.719, E3 +113308.590}
SPL {X  -135.682, Y  +770.527, Z    +0.000, E1   -68.337, E3 +113313.973}
SPL {X  -132.359, Y  +775.105, Z    +0.000, E1   -67.661, E3 +113320.515}
SPL {X  -128.720, Y  +779.765, Z    +0.000, E1   -67.454, E3 +113324.496}
SPL {X  -116.788, Y  +792.975, Z    +0.000, E1   -71.297, E3 +113316.833}
SPL {X   -64.927, Y  +827.895, Z    +0.000, E1   -57.691, E3 +113442.435}
ENDSPLINE

SPLINE
SPL {X  -111.648, Y  +797.871, Z    +0.000, E1   -60.847, E3 +113639.418}
SPL {X  -149.288, Y  +747.285, Z    +0.000, E1   -46.770, E3 +113635.409}
SPL {X  -161.496, Y  +712.364, Z    +0.000, E1   -31.137, E3 +113641.204}
SPL {X  -164.701, Y  +693.202, Z    +0.000, E1   -17.512, E3 +113640.178}
SPL {X  -165.594, Y  +679.817, Z    +0.000, E1    -6.204, E3 +113639.569}
SPL {X  -165.650, Y  +673.522, Z    +0.000, E1    -0.038, E3 +113638.538}
SPL {X  -165.650, Y  +671.354, Z    +0.000, E1    +3.728, E3 +113638.026}
SPL {X  -165.650, Y  +666.485, Z    +0.000, E1   +14.169, E3 +113637.753}
SPL {X  -165.650, Y  +661.236, Z    +0.000, E1   +26.072, E3 +113637.442}
SPL {X  -165.650, Y  +653.063, Z    +0.000, E1   +42.395, E3 +113636.846}
SPL {X  -165.650, Y  +640.535, Z    +0.000, E1   +60.776, E3 +113634.331}
SPL {X  -165.650, Y  +618.963, Z    +0.000, E1   +72.815, E3 +113634.310}
SPL {X  -165.650, Y  +575.208, Z    +0.000, E1   +76.222, E3 +113645.571}
SPL {X  -165.650, Y  +394.754, Z    +0.000, E1   +73.248, E3 +113740.717}
ENDSPLINE

SPLINE
SPL {X  -165.650, Y  +407.500, Z    +0.000, E1   +70.919, E3 +113755.338}
ENDSPLINE

SPLINE
SPL {X  -165.650, Y  +390.855, Z    +0.000, E1   +71.004, E3 +113766.266}
SPL {X  -165.534, Y  +372.295, Z    +0.000, E1   +71.066, E3 +113778.816}
SPL {X  -164.039, Y  +355.451, Z    +0.000, E1   +70.703, E3 +113794.215}
SPL {X  -161.297, Y  +340.777, Z    +0.000, E1   +70.794, E3 +113803.507}
ENDSPLINE

SPLINE
SPL {X  -162.352, Y  +345.609, Z    +0.000, E1   +69.290, E3 +113813.440}
ENDSPLINE

SPLINE
SPL {X  -157.663, Y  +327.685, Z    +0.000, E1   +69.808, E3 +113822.300}
SPL {X  -152.892, Y  +314.750, Z    +0.000, E1   +69.675, E3 +113832.516}
SPL {X  -149.246, Y  +306.628, Z    +0.000, E1   +69.029, E3 +113842.984}
SPL {X  -145.495, Y  +299.310, Z    +0.000, E1   +68.659, E3 +113850.593}
SPL {X  -142.111, Y  +293.387, Z    +0.000, E1   +68.421, E3 +113856.234}
SPL {X  -138.525, Y  +287.667, Z    +0.000, E1   +67.662, E3 +113864.794}
SPL {X  -134.450, Y  +281.737, Z    +0.000, E1   +67.268, E3 +113870.899}
SPL {X  -131.812, Y  +278.173, Z    +0.000, E1   +66.669, E3 +113876.248}
SPL {X  -128.148, Y  +273.533, Z    +0.000, E1   +67.328, E3 +113876.606}
SPL {X  -116.216, Y  +260.459, Z    +0.000, E1   +70.200, E3 +113872.913}
SPL {X   -66.125, Y  +226.621, Z    +0.000, E1   +55.862, E3 +114035.811}
ENDSPLINE

SPLINE
SPL {X  -111.531, Y  +256.023, Z    +0.000, E1   +58.853, E3 +114178.693}
SPL {X  -139.240, Y  +288.767, Z    +0.000, E1   +52.898, E3 +114188.866}
SPL {X  -156.827, Y  +325.161, Z    +0.000, E1   +39.042, E3 +114187.235}
SPL {X  -162.324, Y  +345.471, Z    +0.000, E1   +27.849, E3 +114187.704}
SPL {X  -164.696, Y  +360.744, Z    +0.000, E1   +17.229, E3 +114188.618}
SPL {X  -165.561, Y  +373.081, Z    +0.000, E1    +6.973, E3 +114187.362}
SPL {X  -165.650, Y  +380.800, Z    +0.000, E1    -0.199, E3 +114186.108}
SPL {X  -165.650, Y  +385.044, Z    +0.000, E1    -8.496, E3 +114185.477}
SPL {X  -165.650, Y  +390.492, Z    +0.000, E1   -20.084, E3 +114185.131}
SPL {X  -165.650, Y  +400.081, Z    +0.000, E1   -39.836, E3 +114184.436}
SPL {X  -165.650, Y  +416.111, Z    +0.000, E1   -60.729, E3 +114183.270}
SPL {X  -165.650, Y  +457.077, Z    +0.000, E1   -75.210, E3 +114186.594}
SPL {X  -165.650, Y  +475.293, Z    +0.000, E1   -75.741, E3 +114192.372}
SPL {X  -164.204, Y  +697.342, Z    +0.000, E1   -76.015, E3 +114279.346}
ENDSPLINE

SPLINE
SPL {X  -165.650, Y  +656.030, Z    +0.000, E1   -71.686, E3 +114300.786}
ENDSPLINE

SPLINE
SPL {X  -165.472, Y  +683.167, Z    +0.000, E1   -72.022, E3 +114315.794}
SPL {X  -163.865, Y  +699.752, Z    +0.000, E1   -71.643, E3 +114330.417}
SPL {X  -161.571, Y  +712.032, Z    +0.000, E1   -71.595, E3 +114339.010}
SPL {X  -159.776, Y  +719.221, Z    +0.000, E1   -71.038, E3 +114349.065}
SPL {X  -155.811, Y  +731.738, Z    +0.000, E1   -70.890, E3 +114358.753}
SPL {X  -152.643, Y  +739.844, Z    +0.000, E1   -70.463, E3 +114367.613}
SPL {X  -149.782, Y  +746.247, Z    +0.000, E1   -70.149, E3 +114374.302}
SPL {X  -146.450, Y  +752.910, Z    +0.000, E1   -69.680, E3 +114382.181}
SPL {X  -143.017, Y  +759.082, Z    +0.000, E1   -69.156, E3 +114389.792}
SPL {X  -139.030, Y  +765.558, Z    +0.000, E1   -68.719, E3 +114396.825}
SPL {X  -135.682, Y  +770.527, Z    +0.000, E1   -68.337, E3 +114402.208}
SPL {X  -132.359, Y  +775.105, Z    +0.000, E1   -67.661, E3 +114408.750}
SPL {X  -128.720, Y  +779.765, Z    +0.000, E1   -67.454, E3 +114412.731}
SPL {X  -116.788, Y  +792.975, Z    +0.000, E1   -71.297, E3 +114405.068}
SPL {X   -64.927, Y  +827.895, Z    +0.000, E1   -57.691, E3 +114530.671}
ENDSPLINE

SPLINE
SPL {X  -111.648, Y  +797.871, Z    +0.000, E1   -60.847, E3 +114727.653}
SPL {X  -149.288, Y  +747.285, Z    +0.000, E1   -46.770, E3 +114723.644}
SPL {X  -159.627, Y  +719.761, Z    +0.000, E1   -35.247, E3 +114728.709}
SPL {X  -164.185, Y  +697.485, Z    +0.000, E1   -20.950, E3 +114729.028}
SPL {X  -165.453, Y  +683.578, Z    +0.000, E1    -9.445, E3 +114727.615}
SPL {X  -165.642, Y  +677.105, Z    +0.000, E1    -3.559, E3 +114727.926}
SPL {X  -165.650, Y  +673.522, Z    +0.000, E1    -0.038, E3 +114726.773}
SPL {X  -165.650, Y  +671.354, Z    +0.000, E1    +3.728, E3 +114726.261}
SPL {X  -165.650, Y  +666.485, Z    +0.000, E1   +14.169, E3 +114725.988}
SPL {X  -165.650, Y  +661.236, Z    +0.000, E1   +26.072, E3 +114725.677}
SPL {X  -165.650, Y  +655.357, Z    +0.000, E1   +38.693, E3 +114724.905}
SPL {X  -165.650, Y  +646.637, Z    +0.000, E1   +52.169, E3 +114724.687}
SPL {X  -165.650, Y  +637.909, Z    +0.000, E1   +64.161, E3 +114721.482}
SPL {X  -165.650, Y  +618.963, Z    +0.000, E1   +72.815, E3 +114722.545}
SPL {X  -165.650, Y  +582.897, Z    +0.000, E1   +76.147, E3 +114731.206}
SPL {X  -165.650, Y  +558.388, Z    +0.000, E1   +76.294, E3 +114739.519}
SPL {X  -165.650, Y  +391.690, Z    +0.000, E1   +75.504, E3 +114809.285}
ENDSPLINE

SPLINE
SPL {X  -165.650, Y  +396.283, Z    +0.000, E1   +72.775, E3 +114832.590}
SPL {X  -165.650, Y  +407.500, Z    +0.000, E1   +70.919, E3 +114843.574}
ENDSPLINE

SPLINE
SPL {X  -165.650, Y  +390.855, Z    +0.000, E1   +71.004, E3 +114854.501}
SPL {X  -165.534, Y  +372.295, Z    +0.000, E1   +71.066, E3 +114867.052}
SPL {X  -164.039, Y  +355.451, Z    +0.000, E1   +70.703, E3 +114882.450}
SPL {X  -161.297, Y  +340.777, Z    +0.000, E1   +70.794, E3 +114891.742}
ENDSPLINE

SPLINE
SPL {X  -162.352, Y  +345.609, Z    +0.000, E1   +69.290, E3 +114901.675}
ENDSPLINE

SPLINE
SPL {X  -159.253, Y  +332.909, Z    +0.000, E1   +69.652, E3 +114908.022}
SPL {X  -156.309, Y  +323.661, Z    +0.000, E1   +69.908, E3 +114912.536}
SPL {X  -152.892, Y  +314.750, Z    +0.000, E1   +69.675, E3 +114920.751}
SPL {X  -149.246, Y  +306.628, Z    +0.000, E1   +69.029, E3 +114931.219}
SPL {X  -144.614, Y  +297.712, Z    +0.000, E1   +68.717, E3 +114939.573}
SPL {X  -141.011, Y  +291.576, Z    +0.000, E1   +68.040, E3 +114948.051}
SPL {X  -137.649, Y  +286.345, Z    +0.000, E1   +67.498, E3 +114954.744}
SPL {X  -134.450, Y  +281.737, Z    +0.000, E1   +67.268, E3 +114959.135}
SPL {X  -131.812, Y  +278.173, Z    +0.000, E1   +66.669, E3 +114964.483}
SPL {X  -128.148, Y  +273.533, Z    +0.000, E1   +67.328, E3 +114964.842}
SPL {X  -116.216, Y  +260.459, Z    +0.000, E1   +70.200, E3 +114961.148}
SPL {X   -66.125, Y  +226.621, Z    +0.000, E1   +55.862, E3 +115124.046}
ENDSPLINE

SPLINE
SPL {X  -111.531, Y  +256.023, Z    +0.000, E1   +58.853, E3 +115266.928}
SPL {X  -139.240, Y  +288.767, Z    +0.000, E1   +52.898, E3 +115277.101}
SPL {X  -156.827, Y  +325.161, Z    +0.000, E1   +39.042, E3 +115275.470}
SPL {X  -162.324, Y  +345.471, Z    +0.000, E1   +27.849, E3 +115275.939}
SPL {X  -164.696, Y  +360.744, Z    +0.000, E1   +17.229, E3 +115276.853}
SPL {X  -165.561, Y  +373.081, Z    +0.000, E1    +6.973, E3 +115275.597}
SPL {X  -165.650, Y  +379.105, Z    +0.000, E1    +1.379, E3 +115275.158}
SPL {X  -165.650, Y  +380.899, Z    +0.000, E1    -0.394, E3 +115274.296}
SPL {X  -165.650, Y  +385.044, Z    +0.000, E1    -8.496, E3 +115273.712}
SPL {X  -165.650, Y  +388.717, Z    +0.000, E1   -16.400, E3 +115273.568}
SPL {X  -165.650, Y  +394.613, Z    +0.000, E1   -29.184, E3 +115273.037}
SPL {X  -165.650, Y  +402.836, Z    +0.000, E1   -44.797, E3 +115272.439}
SPL {X  -165.650, Y  +416.111, Z    +0.000, E1   -60.729, E3 +115271.506}
SPL {X  -165.650, Y  +457.077, Z    +0.000, E1   -75.210, E3 +115274.829}
SPL {X  -165.650, Y  +475.293, Z    +0.000, E1   -75.741, E3 +115280.607}
SPL {X  -164.204, Y  +697.342, Z    +0.000, E1   -76.015, E3 +115367.582}
ENDSPLINE

SPLINE
SPL {X  -165.650, Y  +664.340, Z    +0.000, E1   -71.862, E3 +115392.985}
ENDSPLINE

SPLINE
SPL {X  -165.237, Y  +687.187, Z    +0.000, E1   -71.947, E3 +115407.247}
SPL {X  -163.865, Y  +699.752, Z    +0.000, E1   -71.643, E3 +115418.653}
SPL {X  -161.821, Y  +710.908, Z    +0.000, E1   -71.322, E3 +115429.193}
SPL {X  -158.993, Y  +721.987, Z    +0.000, E1   -71.173, E3 +115437.981}
SPL {X  -155.811, Y  +731.738, Z    +0.000, E1   -70.890, E3 +115446.989}
SPL {X  -152.643, Y  +739.844, Z    +0.000, E1   -70.463, E3 +115455.848}
SPL {X  -149.782, Y  +746.247, Z    +0.000, E1   -70.149, E3 +115462.538}
SPL {X  -146.450, Y  +752.910, Z    +0.000, E1   -69.680, E3 +115470.416}
SPL {X  -143.017, Y  +759.082, Z    +0.000, E1   -69.156, E3 +115478.027}
SPL {X  -139.030, Y  +765.558, Z    +0.000, E1   -68.719, E3 +115485.060}
SPL {X  -134.589, Y  +772.070, Z    +0.000, E1   -68.090, E3 +115492.909}
SPL {X  -129.830, Y  +778.379, Z    +0.000, E1   -67.491, E3 +115499.919}
SPL {X  -116.788, Y  +792.975, Z    +0.000, E1   -71.297, E3 +115493.303}
SPL {X   -64.927, Y  +827.895, Z    +0.000, E1   -57.691, E3 +115618.906}
ENDSPLINE

SPLINE
SPL {X  -111.648, Y  +797.871, Z    +0.000, E1   -60.847, E3 +115815.889}
SPL {X  -149.288, Y  +747.285, Z    +0.000, E1   -46.770, E3 +115811.879}
SPL {X  -159.627, Y  +719.761, Z    +0.000, E1   -35.247, E3 +115816.944}
SPL {X  -164.185, Y  +697.485, Z    +0.000, E1   -20.950, E3 +115817.263}
SPL {X  -165.594, Y  +679.817, Z    +0.000, E1    -6.204, E3 +115816.040}
SPL {X  -165.650, Y  +673.522, Z    +0.000, E1    -0.038, E3 +115815.009}
SPL {X  -165.650, Y  +671.354, Z    +0.000, E1    +3.728, E3 +115814.496}
SPL {X  -165.650, Y  +666.485, Z    +0.000, E1   +14.169, E3 +115814.223}
SPL {X  -165.650, Y  +661.236, Z    +0.000, E1   +26.072, E3 +115813.913}
SPL {X  -165.650, Y  +653.063, Z    +0.000, E1   +42.395, E3 +115813.317}
SPL {X  -165.650, Y  +640.535, Z    +0.000, E1   +60.776, E3 +115810.801}
SPL {X  -165.650, Y  +618.963, Z    +0.000, E1   +72.815, E3 +115810.780}
SPL {X  -165.650, Y  +575.208, Z    +0.000, E1   +76.222, E3 +115822.041}
SPL {X  -165.650, Y  +394.754, Z    +0.000, E1   +73.248, E3 +115917.188}
ENDSPLINE

SPLINE
SPL {X  -165.650, Y  +407.500, Z    +0.000, E1   +70.919, E3 +115931.809}
ENDSPLINE

SPLINE
SPL {X  -165.650, Y  +390.855, Z    +0.000, E1   +71.004, E3 +115942.737}
SPL {X  -165.534, Y  +372.295, Z    +0.000, E1   +71.066, E3 +115955.287}
SPL {X  -164.687, Y  +360.663, Z    +0.000, E1   +70.826, E3 +115965.579}
SPL {X  -162.841, Y  +348.123, Z    +0.000, E1   +70.683, E3 +115975.958}
SPL {X  -162.352, Y  +345.609, Z    +0.000, E1   +69.290, E3 +115989.911}
SPL {X  -159.253, Y  +332.909, Z    +0.000, E1   +69.652, E3 +115996.257}
SPL {X  -155.267, Y  +320.775, Z    +0.000, E1   +69.854, E3 +116003.350}
SPL {X  -151.256, Y  +310.961, Z    +0.000, E1   +69.467, E3 +116013.225}
SPL {X  -148.628, Y  +305.359, Z    +0.000, E1   +68.848, E3 +116021.504}
SPL {X  -144.614, Y  +297.712, Z    +0.000, E1   +68.717, E3 +116027.808}
SPL {X  -141.011, Y  +291.576, Z    +0.000, E1   +68.040, E3 +116036.286}
SPL {X  -137.649, Y  +286.345, Z    +0.000, E1   +67.498, E3 +116042.980}
SPL {X  -134.450, Y  +281.737, Z    +0.000, E1   +67.268, E3 +116047.370}
SPL {X  -131.812, Y  +278.173, Z    +0.000, E1   +66.669, E3 +116052.718}
SPL {X  -128.148, Y  +273.533, Z    +0.000, E1   +67.328, E3 +116053.077}
SPL {X  -116.216, Y  +260.459, Z    +0.000, E1   +70.200, E3 +116049.383}
SPL {X   -66.125, Y  +226.621, Z    +0.000, E1   +55.862, E3 +116212.282}
ENDSPLINE

SPLINE
SPL {X  -111.531, Y  +256.023, Z    +0.000, E1   +58.853, E3 +116355.163}
SPL {X  -139.240, Y  +288.767, Z    +0.000, E1   +52.898, E3 +116365.336}
SPL {X  -156.827, Y  +325.161, Z    +0.000, E1   +39.042, E3 +116363.706}
SPL {X  -162.324, Y  +345.471, Z    +0.000, E1   +27.849, E3 +116364.174}
SPL {X  -165.055, Y  +364.477, Z    +0.000, E1   +14.326, E3 +116364.612}
SPL {X  -165.646, Y  +377.353, Z    +0.000, E1    +3.112, E3 +116363.569}
SPL {X  -165.650, Y  +380.500, Z    +0.000, E1    -0.000, E3 +116362.695}
SPL {X  -165.650, Y  +381.828, Z    +0.000, E1    -2.219, E3 +116362.148}
SPL {X  -165.650, Y  +385.044, Z    +0.000, E1    -8.496, E3 +116361.947}
SPL {X  -165.650, Y  +388.717, Z    +0.000, E1   -16.400, E3 +116361.803}
SPL {X  -165.650, Y  +394.613, Z    +0.000, E1   -29.184, E3 +116361.272}
SPL {X  -165.650, Y  +402.836, Z    +0.000, E1   -44.797, E3 +116360.674}
SPL {X  -165.650, Y  +416.111, Z    +0.000, E1   -60.729, E3 +116359.741}
SPL {X  -165.650, Y  +471.994, Z    +0.000, E1   -75.670, E3 +116367.794}
SPL {X  -164.204, Y  +697.342, Z    +0.000, E1   -76.015, E3 +116455.817}
ENDSPLINE

SPLINE
SPL {X  -165.650, Y  +664.340, Z    +0.000, E1   -71.862, E3 +116481.221}
ENDSPLINE

SPLINE
SPL {X  -165.237, Y  +687.187, Z    +0.000, E1   -71.947, E3 +116495.482}
SPL {X  -163.865, Y  +699.752, Z    +0.000, E1   -71.643, E3 +116506.888}
SPL {X  -161.041, Y  +714.304, Z    +0.000, E1   -71.423, E3 +116518.791}
SPL {X  -159.124, Y  +721.538, Z    +0.000, E1   -70.872, E3 +116528.444}
SPL {X  -155.811, Y  +731.738, Z    +0.000, E1   -70.890, E3 +116535.224}
SPL {X  -152.643, Y  +739.844, Z    +0.000, E1   -70.463, E3 +116544.083}
SPL {X  -149.782, Y  +746.247, Z    +0.000, E1   -70.149, E3 +116550.773}
SPL {X  -146.450, Y  +752.910, Z    +0.000, E1   -69.680, E3 +116558.651}
SPL {X  -143.017, Y  +759.082, Z    +0.000, E1   -69.156, E3 +116566.262}
SPL {X  -140.057, Y  +763.953, Z    +0.000, E1   -68.829, E3 +116571.502}
SPL {X  -136.535, Y  +769.298, Z    +0.000, E1   -68.442, E3 +116577.363}
SPL {X  -132.359, Y  +775.105, Z    +0.000, E1   -67.661, E3 +116585.221}
SPL {X  -128.720, Y  +779.765, Z    +0.000, E1   -67.454, E3 +116589.202}
SPL {X  -116.788, Y  +792.975, Z    +0.000, E1   -71.297, E3 +116581.538}
SPL {X   -64.927, Y  +827.895, Z    +0.000, E1   -57.691, E3 +116707.141}
ENDSPLINE

SPLINE
SPL {X  -111.648, Y  +797.871, Z    +0.000, E1   -60.847, E3 +116904.124}
SPL {X  -149.288, Y  +747.285, Z    +0.000, E1   -46.770, E3 +116900.115}
SPL {X  -161.496, Y  +712.364, Z    +0.000, E1   -31.137, E3 +116905.910}
SPL {X  -164.701, Y  +693.202, Z    +0.000, E1   -17.512, E3 +116904.884}
SPL {X  -165.453, Y  +683.578, Z    +0.000, E1    -9.445, E3 +116904.086}
SPL {X  -165.642, Y  +677.105, Z    +0.000, E1    -3.559, E3 +116904.396}
SPL {X  -165.650, Y  +673.263, Z    +0.000, E1    +0.216, E3 +116903.156}
SPL {X  -165.650, Y  +670.095, Z    +0.000, E1    +6.482, E3 +116902.560}
SPL {X  -165.650, Y  +666.485, Z    +0.000, E1   +14.169, E3 +116902.459}
SPL {X  -165.650, Y  +661.236, Z    +0.000, E1   +26.072, E3 +116902.148}
SPL {X  -165.650, Y  +653.063, Z    +0.000, E1   +42.395, E3 +116901.552}
SPL {X  -165.650, Y  +640.535, Z    +0.000, E1   +60.776, E3 +116899.037}
SPL {X  -165.650, Y  +618.963, Z    +0.000, E1   +72.815, E3 +116899.016}
SPL {X  -165.650, Y  +575.208, Z    +0.000, E1   +76.222, E3 +116910.277}
SPL {X  -165.650, Y  +394.754, Z    +0.000, E1   +73.248, E3 +117005.423}
ENDSPLINE

SPLINE
SPL {X  -165.650, Y  +407.500, Z    +0.000, E1   +70.919, E3 +117020.044}
ENDSPLINE

SPLINE
SPL {X  -165.650, Y  +390.855, Z    +0.000, E1   +71.004, E3 +117030.972}
SPL {X  -165.534, Y  +372.295, Z    +0.000, E1   +71.066, E3 +117043.522}
SPL {X  -164.039, Y  +355.451, Z    +0.000, E1   +70.703, E3 +117058.920}
SPL {X  -161.297, Y  +340.777, Z    +0.000, E1   +70.794, E3 +117068.213}
ENDSPLINE

SPLINE
SPL {X  -162.352, Y  +345.609, Z    +0.000, E1   +69.290, E3 +117078.146}
ENDSPLINE

SPLINE
SPL {X  -157.663, Y  +327.685, Z    +0.000, E1   +69.808, E3 +117087.006}
SPL {X  -154.072, Y  +317.659, Z    +0.000, E1   +69.748, E3 +117094.498}
SPL {X  -151.256, Y  +310.961, Z    +0.000, E1   +69.467, E3 +117101.461}
SPL {X  -148.628, Y  +305.359, Z    +0.000, E1   +68.848, E3 +117109.739}
SPL {X  -145.495, Y  +299.310, Z    +0.000, E1   +68.659, E3 +117115.299}
SPL {X  -141.249, Y  +291.963, Z    +0.000, E1   +68.223, E3 +117123.279}
SPL {X  -137.649, Y  +286.345, Z    +0.000, E1   +67.498, E3 +117131.215}
SPL {X  -134.450, Y  +281.737, Z    +0.000, E1   +67.268, E3 +117135.605}
SPL {X  -131.812, Y  +278.173, Z    +0.000, E1   +66.669, E3 +117140.954}
SPL {X  -128.148, Y  +273.533, Z    +0.000, E1   +67.328, E3 +117141.312}
SPL {X  -116.216, Y  +260.459, Z    +0.000, E1   +70.200, E3 +117137.619}
SPL {X   -66.125, Y  +226.621, Z    +0.000, E1   +55.862, E3 +117300.517}
ENDSPLINE

SPLINE
SPL {X  -111.531, Y  +256.023, Z    +0.000, E1   +58.853, E3 +117443.399}
SPL {X  -139.240, Y  +288.767, Z    +0.000, E1   +52.898, E3 +117453.572}
SPL {X  -156.827, Y  +325.161, Z    +0.000, E1   +39.042, E3 +117451.941}
SPL {X  -162.324, Y  +345.471, Z    +0.000, E1   +27.849, E3 +117452.410}
SPL {X  -164.696, Y  +360.744, Z    +0.000, E1   +17.229, E3 +117453.324}
SPL {X  -165.561, Y  +373.081, Z    +0.000, E1    +6.973, E3 +117452.068}
SPL {X  -165.650, Y  +379.105, Z    +0.000, E1    +1.379, E3 +117451.629}
SPL {X  -165.650, Y  +380.899, Z    +0.000, E1    -0.394, E3 +117450.766}
SPL {X  -165.650, Y  +385.044, Z    +0.000, E1    -8.496, E3 +117450.183}
SPL {X  -165.650, Y  +390.492, Z    +0.000, E1   -20.084, E3 +117449.837}
SPL {X  -165.650, Y  +400.081, Z    +0.000, E1   -39.836, E3 +117449.142}
SPL {X  -165.650, Y  +416.111, Z    +0.000, E1   -60.729, E3 +117447.976}
SPL {X  -165.650, Y  +457.077, Z    +0.000, E1   -75.210, E3 +117451.300}
SPL {X  -165.650, Y  +475.293, Z    +0.000, E1   -75.741, E3 +117457.078}
SPL {X  -164.204, Y  +697.342, Z    +0.000, E1   -76.015, E3 +117544.052}
ENDSPLINE

SPLINE
SPL {X  -165.650, Y  +656.030, Z    +0.000, E1   -71.686, E3 +117565.492}
ENDSPLINE

SPLINE
SPL {X  -165.610, Y  +679.119, Z    +0.000, E1   -71.889, E3 +117579.115}
SPL {X  -163.827, Y  +700.009, Z    +0.000, E1   -71.824, E3 +117593.681}
SPL {X  -161.821, Y  +710.908, Z    +0.000, E1   -71.322, E3 +117605.663}
SPL {X  -158.993, Y  +721.987, Z    +0.000, E1   -71.173, E3 +117614.452}
SPL {X  -155.811, Y  +731.738, Z    +0.000, E1   -70.890, E3 +117623.459}
SPL {X  -152.643, Y  +739.844, Z    +0.000, E1   -70.463, E3 +117632.319}
SPL {X  -149.782, Y  +746.247, Z    +0.000, E1   -70.149, E3 +117639.008}
SPL {X  -146.450, Y  +752.910, Z    +0.000, E1   -69.680, E3 +117646.886}
SPL {X  -143.017, Y  +759.082, Z    +0.000, E1   -69.156, E3 +117654.498}
SPL {X  -139.030, Y  +765.558, Z    +0.000, E1   -68.719, E3 +117661.531}
SPL {X  -134.589, Y  +772.070, Z    +0.000, E1   -68.090, E3 +117669.380}
SPL {X  -129.830, Y  +778.379, Z    +0.000, E1   -67.491, E3 +117676.389}
SPL {X  -116.788, Y  +792.975, Z    +0.000, E1   -71.297, E3 +117669.774}
SPL {X   -64.927, Y  +827.895, Z    +0.000, E1   -57.691, E3 +117795.377}
ENDSPLINE

SPLINE
SPL {X  -111.648, Y  +797.871, Z    +0.000, E1   -60.847, E3 +117992.359}
SPL {X  -149.288, Y  +747.285, Z    +0.000, E1   -46.770, E3 +117988.350}
SPL {X  -159.627, Y  +719.761, Z    +0.000, E1   -35.247, E3 +117993.415}
SPL {X  -164.185, Y  +697.485, Z    +0.000, E1   -20.950, E3 +117993.734}
SPL {X  -165.594, Y  +679.817, Z    +0.000, E1    -6.204, E3 +117992.510}
SPL {X  -165.650, Y  +673.522, Z    +0.000, E1    -0.038, E3 +117991.479}
SPL {X  -165.650, Y  +671.354, Z    +0.000, E1    +3.728, E3 +117990.967}
SPL {X  -165.650, Y  +666.485, Z    +0.000, E1   +14.169, E3 +117990.694}
SPL {X  -165.650, Y  +661.236, Z    +0.000, E1   +26.072, E3 +117990.383}
SPL {X  -165.650, Y  +653.063, Z    +0.000, E1   +42.395, E3 +117989.787}
SPL {X  -165.650, Y  +640.535, Z    +0.000, E1   +60.776, E3 +117987.272}
SPL {X  -165.650, Y  +618.963, Z    +0.000, E1   +72.815, E3 +117987.251}
SPL {X  -165.650, Y  +575.208, Z    +0.000, E1   +76.222, E3 +117998.512}
SPL {X  -165.650, Y  +394.754, Z    +0.000, E1   +73.248, E3 +118093.658}
ENDSPLINE

SPLINE
SPL {X  -165.650, Y  +407.500, Z    +0.000, E1   +70.919, E3 +118108.279}
ENDSPLINE

SPLINE
SPL {X  -165.650, Y  +390.855, Z    +0.000, E1   +71.004, E3 +118119.207}
SPL {X  -165.534, Y  +372.295, Z    +0.000, E1   +71.066, E3 +118131.758}
SPL {X  -164.687, Y  +360.663, Z    +0.000, E1   +70.826, E3 +118142.049}
SPL {X  -162.841, Y  +348.123, Z    +0.000, E1   +70.683, E3 +118152.428}
SPL {X  -162.352, Y  +345.609, Z    +0.000, E1   +69.290, E3 +118166.381}
SPL {X  -159.253, Y  +332.909, Z    +0.000, E1   +69.652, E3 +118172.728}
SPL {X  -155.267, Y  +320.775, Z    +0.000, E1   +69.854, E3 +118179.821}
SPL {X  -151.256, Y  +310.961, Z    +0.000, E1   +69.467, E3 +118189.696}
SPL {X  -148.628, Y  +305.359, Z    +0.000, E1   +68.848, E3 +118197.974}
SPL {X  -144.614, Y  +297.712, Z    +0.000, E1   +68.717, E3 +118204.279}
SPL {X  -141.011, Y  +291.576, Z    +0.000, E1   +68.040, E3 +118212.757}
SPL {X  -137.649, Y  +286.345, Z    +0.000, E1   +67.498, E3 +118219.450}
SPL {X  -134.450, Y  +281.737, Z    +0.000, E1   +67.268, E3 +118223.840}
SPL {X  -131.812, Y  +278.173, Z    +0.000, E1   +66.669, E3 +118229.189}
SPL {X  -128.148, Y  +273.533, Z    +0.000, E1   +67.328, E3 +118229.547}
SPL {X  -116.216, Y  +260.459, Z    +0.000, E1   +70.200, E3 +118225.854}
SPL {X   -66.125, Y  +226.621, Z    +0.000, E1   +55.862, E3 +118388.752}
ENDSPLINE

SPLINE
SPL {X  -111.531, Y  +256.023, Z    +0.000, E1   +58.853, E3 +118531.634}
SPL {X  -139.240, Y  +288.767, Z    +0.000, E1   +52.898, E3 +118541.807}
SPL {X  -156.827, Y  +325.161, Z    +0.000, E1   +39.042, E3 +118540.176}
SPL {X  -162.324, Y  +345.471, Z    +0.000, E1   +27.849, E3 +118540.645}
SPL {X  -165.055, Y  +364.477, Z    +0.000, E1   +14.326, E3 +118541.083}
SPL {X  -165.646, Y  +377.353, Z    +0.000, E1    +3.112, E3 +118540.040}
SPL {X  -165.650, Y  +380.500, Z    +0.000, E1    -0.000, E3 +118539.166}
SPL {X  -165.650, Y  +381.828, Z    +0.000, E1    -2.219, E3 +118538.618}
SPL {X  -165.650, Y  +385.044, Z    +0.000, E1    -8.496, E3 +118538.418}
SPL {X  -165.650, Y  +388.717, Z    +0.000, E1   -16.400, E3 +118538.274}
SPL {X  -165.650, Y  +394.613, Z    +0.000, E1   -29.184, E3 +118537.742}
SPL {X  -165.650, Y  +402.836, Z    +0.000, E1   -44.797, E3 +118537.145}
SPL {X  -165.650, Y  +416.111, Z    +0.000, E1   -60.729, E3 +118536.212}
SPL {X  -165.650, Y  +471.994, Z    +0.000, E1   -75.670, E3 +118544.265}
SPL {X  -164.204, Y  +697.342, Z    +0.000, E1   -76.015, E3 +118632.288}
ENDSPLINE

SPLINE
SPL {X  -165.650, Y  +664.340, Z    +0.000, E1   -71.862, E3 +118657.691}
ENDSPLINE

SPLINE
SPL {X  -165.237, Y  +687.187, Z    +0.000, E1   -71.947, E3 +118671.953}
SPL {X  -163.865, Y  +699.752, Z    +0.000, E1   -71.643, E3 +118683.358}
SPL {X  -161.041, Y  +714.304, Z    +0.000, E1   -71.423, E3 +118695.262}
SPL {X  -159.124, Y  +721.538, Z    +0.000, E1   -70.872, E3 +118704.914}
SPL {X  -155.811, Y  +731.738, Z    +0.000, E1   -70.890, E3 +118711.695}
SPL {X  -152.643, Y  +739.844, Z    +0.000, E1   -70.463, E3 +118720.554}
SPL {X  -149.782, Y  +746.247, Z    +0.000, E1   -70.149, E3 +118727.244}
SPL {X  -146.450, Y  +752.910, Z    +0.000, E1   -69.680, E3 +118735.122}
SPL {X  -143.017, Y  +759.082, Z    +0.000, E1   -69.156, E3 +118742.733}
SPL {X  -139.030, Y  +765.558, Z    +0.000, E1   -68.719, E3 +118749.766}
SPL {X  -134.589, Y  +772.070, Z    +0.000, E1   -68.090, E3 +118757.615}
SPL {X  -129.830, Y  +778.379, Z    +0.000, E1   -67.491, E3 +118764.625}
SPL {X  -116.788, Y  +792.975, Z    +0.000, E1   -71.297, E3 +118758.009}
SPL {X   -64.927, Y  +827.895, Z    +0.000, E1   -57.691, E3 +118883.612}
ENDSPLINE

SPLINE
SPL {X  -111.648, Y  +797.871, Z    +0.000, E1   -60.847, E3 +119080.594}
SPL {X  -149.288, Y  +747.285, Z    +0.000, E1   -46.770, E3 +119076.585}
SPL {X  -159.627, Y  +719.761, Z    +0.000, E1   -35.247, E3 +119081.650}
SPL {X  -164.185, Y  +697.485, Z    +0.000, E1   -20.950, E3 +119081.969}
SPL {X  -165.594, Y  +679.817, Z    +0.000, E1    -6.204, E3 +119080.746}
SPL {X  -165.650, Y  +673.522, Z    +0.000, E1    -0.038, E3 +119079.715}
SPL {X  -165.650, Y  +671.354, Z    +0.000, E1    +3.728, E3 +119079.202}
SPL {X  -165.650, Y  +666.485, Z    +0.000, E1   +14.169, E3 +119078.929}
SPL {X  -165.650, Y  +661.236, Z    +0.000, E1   +26.072, E3 +119078.618}
SPL {X  -165.650, Y  +653.063, Z    +0.000, E1   +42.395, E3 +119078.023}
SPL {X  -165.650, Y  +640.535, Z    +0.000, E1   +60.776, E3 +119075.507}
SPL {X  -165.650, Y  +618.963, Z    +0.000, E1   +72.815, E3 +119075.486}
SPL {X  -165.650, Y  +575.208, Z    +0.000, E1   +76.222, E3 +119086.747}
SPL {X  -165.650, Y  +394.754, Z    +0.000, E1   +73.248, E3 +119181.894}
ENDSPLINE

SPLINE
SPL {X  -165.650, Y  +407.500, Z    +0.000, E1   +70.919, E3 +119196.515}
ENDSPLINE

SPLINE
SPL {X  -165.650, Y  +390.855, Z    +0.000, E1   +71.004, E3 +119207.442}
SPL {X  -165.534, Y  +372.295, Z    +0.000, E1   +71.066, E3 +119219.993}
SPL {X  -164.687, Y  +360.663, Z    +0.000, E1   +70.826, E3 +119230.285}
SPL {X  -162.841, Y  +348.123, Z    +0.000, E1   +70.683, E3 +119240.663}
SPL {X  -162.352, Y  +345.609, Z    +0.000, E1   +69.290, E3 +119254.617}
SPL {X  -157.663, Y  +327.685, Z    +0.000, E1   +69.808, E3 +119263.477}
SPL {X  -154.072, Y  +317.659, Z    +0.000, E1   +69.748, E3 +119270.968}
SPL {X  -151.256, Y  +310.961, Z    +0.000, E1   +69.467, E3 +119277.931}
SPL {X  -148.628, Y  +305.359, Z    +0.000, E1   +68.848, E3 +119286.210}
SPL {X  -145.495, Y  +299.310, Z    +0.000, E1   +68.659, E3 +119291.769}
SPL {X  -142.111, Y  +293.387, Z    +0.000, E1   +68.421, E3 +119297.411}
SPL {X  -138.525, Y  +287.667, Z    +0.000, E1   +67.662, E3 +119305.970}
SPL {X  -134.450, Y  +281.737, Z    +0.000, E1   +67.268, E3 +119312.076}
SPL {X  -131.812, Y  +278.173, Z    +0.000, E1   +66.669, E3 +119317.424}
SPL {X  -128.148, Y  +273.533, Z    +0.000, E1   +67.328, E3 +119317.783}
SPL {X  -116.216, Y  +260.459, Z    +0.000, E1   +70.200, E3 +119314.089}
SPL {X   -66.125, Y  +226.621, Z    +0.000, E1   +55.862, E3 +119476.987}
ENDSPLINE

SPLINE
SPL {X  -111.531, Y  +256.023, Z    +0.000, E1   +58.853, E3 +119619.869}
SPL {X  -139.240, Y  +288.767, Z    +0.000, E1   +52.898, E3 +119630.042}
SPL {X  -156.827, Y  +325.161, Z    +0.000, E1   +39.042, E3 +119628.412}
SPL {X  -162.324, Y  +345.471, Z    +0.000, E1   +27.849, E3 +119628.880}
SPL {X  -165.055, Y  +364.477, Z    +0.000, E1   +14.326, E3 +119629.318}
SPL {X  -165.646, Y  +377.353, Z    +0.000, E1    +3.112, E3 +119628.275}
SPL {X  -165.650, Y  +380.899, Z    +0.000, E1    -0.394, E3 +119627.237}
SPL {X  -165.650, Y  +385.044, Z    +0.000, E1    -8.496, E3 +119626.653}
SPL {X  -165.650, Y  +388.717, Z    +0.000, E1   -16.400, E3 +119626.509}
SPL {X  -165.650, Y  +394.613, Z    +0.000, E1   -29.184, E3 +119625.978}
SPL {X  -165.650, Y  +402.836, Z    +0.000, E1   -44.797, E3 +119625.380}
SPL {X  -165.650, Y  +416.111, Z    +0.000, E1   -60.729, E3 +119624.447}
SPL {X  -165.650, Y  +471.994, Z    +0.000, E1   -75.670, E3 +119632.500}
SPL {X  -164.204, Y  +697.342, Z    +0.000, E1   -76.015, E3 +119720.523}
ENDSPLINE

SPLINE
SPL {X  -165.650, Y  +664.340, Z    +0.000, E1   -71.862, E3 +119745.927}
ENDSPLINE

SPLINE
SPL {X  -165.116, Y  +688.792, Z    +0.000, E1   -71.759, E3 +119763.366}
SPL {X  -162.089, Y  +709.665, Z    +0.000, E1   -71.739, E3 +119777.420}
SPL {X  -160.450, Y  +716.681, Z    +0.000, E1   -71.166, E3 +119787.223}
SPL {X  -159.124, Y  +721.538, Z    +0.000, E1   -70.872, E3 +119793.150}
SPL {X  -155.811, Y  +731.738, Z    +0.000, E1   -70.890, E3 +119799.930}
SPL {X  -152.643, Y  +739.844, Z    +0.000, E1   -70.463, E3 +119808.789}
SPL {X  -149.782, Y  +746.247, Z    +0.000, E1   -70.149, E3 +119815.479}
SPL {X  -146.450, Y  +752.910, Z    +0.000, E1   -69.680, E3 +119823.357}
SPL {X  -143.017, Y  +759.082, Z    +0.000, E1   -69.156, E3 +119830.968}
SPL {X  -140.057, Y  +763.953, Z    +0.000, E1   -68.829, E3 +119836.208}
SPL {X  -136.535, Y  +769.298, Z    +0.000, E1   -68.442, E3 +119842.069}
SPL {X  -133.553, Y  +773.498, Z    +0.000, E1   -67.773, E3 +119848.234}
SPL {X  -129.830, Y  +778.379, Z    +0.000, E1   -67.491, E3 +119852.860}
SPL {X  -116.788, Y  +792.975, Z    +0.000, E1   -71.297, E3 +119846.244}
SPL {X   -70.520, Y  +825.390, Z    +0.000, E1   -59.928, E3 +119940.155}
SPL {X   -62.607, Y  +828.863, Z    +0.000, E1   -56.584, E3 +119995.039}
ENDSPLINE

SPLINE
SPL {X  -111.648, Y  +797.871, Z    +0.000, E1   -60.847, E3 +120168.830}
SPL {X  -149.288, Y  +747.285, Z    +0.000, E1   -46.770, E3 +120164.820}
SPL {X  -161.496, Y  +712.364, Z    +0.000, E1   -31.137, E3 +120170.616}
SPL {X  -164.701, Y  +693.202, Z    +0.000, E1   -17.512, E3 +120169.590}
SPL {X  -165.594, Y  +679.817, Z    +0.000, E1    -6.204, E3 +120168.981}
SPL {X  -165.650, Y  +673.522, Z    +0.000, E1    -0.038, E3 +120167.950}
SPL {X  -165.650, Y  +671.354, Z    +0.000, E1    +3.728, E3 +120167.437}
SPL {X  -165.650, Y  +666.485, Z    +0.000, E1   +14.169, E3 +120167.165}
SPL {X  -165.650, Y  +661.236, Z    +0.000, E1   +26.072, E3 +120166.854}
SPL {X  -165.650, Y  +653.063, Z    +0.000, E1   +42.395, E3 +120166.258}
SPL {X  -165.650, Y  +640.535, Z    +0.000, E1   +60.776, E3 +120163.743}
SPL {X  -165.650, Y  +618.963, Z    +0.000, E1   +72.815, E3 +120163.722}
SPL {X  -165.650, Y  +575.208, Z    +0.000, E1   +76.222, E3 +120174.982}
SPL {X  -165.650, Y  +394.754, Z    +0.000, E1   +73.248, E3 +120270.129}
ENDSPLINE

SPLINE
SPL {X  -165.650, Y  +407.500, Z    +0.000, E1   +70.919, E3 +120284.750}
ENDSPLINE

SPLINE
SPL {X  -165.650, Y  +390.855, Z    +0.000, E1   +71.004, E3 +120295.678}
SPL {X  -165.534, Y  +372.295, Z    +0.000, E1   +71.066, E3 +120308.228}
SPL {X  -164.687, Y  +360.663, Z    +0.000, E1   +70.826, E3 +120318.520}
SPL {X  -162.841, Y  +348.123, Z    +0.000, E1   +70.683, E3 +120328.899}
SPL {X  -162.352, Y  +345.609, Z    +0.000, E1   +69.290, E3 +120342.852}
SPL {X  -159.253, Y  +332.909, Z    +0.000, E1   +69.652, E3 +120349.198}
SPL {X  -156.309, Y  +323.661, Z    +0.000, E1   +69.908, E3 +120353.713}
SPL {X  -152.892, Y  +314.750, Z    +0.000, E1   +69.675, E3 +120361.928}
SPL {X  -149.246, Y  +306.628, Z    +0.000, E1   +69.029, E3 +120372.396}
SPL {X  -145.495, Y  +299.310, Z    +0.000, E1   +68.659, E3 +120380.004}
SPL {X  -142.111, Y  +293.387, Z    +0.000, E1   +68.421, E3 +120385.646}
SPL {X  -138.525, Y  +287.667, Z    +0.000, E1   +67.662, E3 +120394.206}
SPL {X  -134.450, Y  +281.737, Z    +0.000, E1   +67.268, E3 +120400.311}
SPL {X  -131.812, Y  +278.173, Z    +0.000, E1   +66.669, E3 +120405.660}
SPL {X  -128.148, Y  +273.533, Z    +0.000, E1   +67.328, E3 +120406.018}
SPL {X  -116.216, Y  +260.459, Z    +0.000, E1   +70.200, E3 +120402.325}
SPL {X   -66.125, Y  +226.621, Z    +0.000, E1   +55.862, E3 +120565.223}
ENDSPLINE

SPLINE
SPL {X  -111.531, Y  +256.023, Z    +0.000, E1   +58.853, E3 +120708.105}
SPL {X  -139.240, Y  +288.767, Z    +0.000, E1   +52.898, E3 +120718.277}
SPL {X  -156.827, Y  +325.161, Z    +0.000, E1   +39.042, E3 +120716.647}
SPL {X  -162.324, Y  +345.471, Z    +0.000, E1   +27.849, E3 +120717.115}
SPL {X  -164.696, Y  +360.744, Z    +0.000, E1   +17.229, E3 +120718.030}
SPL {X  -165.561, Y  +373.081, Z    +0.000, E1    +6.973, E3 +120716.774}
SPL {X  -165.650, Y  +379.105, Z    +0.000, E1    +1.379, E3 +120716.335}
SPL {X  -165.650, Y  +380.899, Z    +0.000, E1    -0.394, E3 +120715.472}
SPL {X  -165.650, Y  +385.044, Z    +0.000, E1    -8.496, E3 +120714.888}
SPL {X  -165.650, Y  +388.717, Z    +0.000, E1   -16.400, E3 +120714.744}
SPL {X  -165.650, Y  +394.613, Z    +0.000, E1   -29.184, E3 +120714.213}
SPL {X  -165.650, Y  +402.836, Z    +0.000, E1   -44.797, E3 +120713.616}
SPL {X  -165.650, Y  +416.111, Z    +0.000, E1   -60.729, E3 +120712.682}
SPL {X  -165.650, Y  +457.077, Z    +0.000, E1   -75.210, E3 +120716.006}
SPL {X  -165.650, Y  +475.293, Z    +0.000, E1   -75.741, E3 +120721.784}
SPL {X  -164.204, Y  +697.342, Z    +0.000, E1   -76.015, E3 +120808.758}
ENDSPLINE

SPLINE
SPL {X  -165.650, Y  +664.340, Z    +0.000, E1   -71.862, E3 +120834.162}
ENDSPLINE

SPLINE
SPL {X  -165.237, Y  +687.187, Z    +0.000, E1   -71.947, E3 +120848.423}
SPL {X  -163.865, Y  +699.752, Z    +0.000, E1   -71.643, E3 +120859.829}
SPL {X  -161.821, Y  +710.908, Z    +0.000, E1   -71.322, E3 +120870.369}
SPL {X  -158.993, Y  +721.987, Z    +0.000, E1   -71.173, E3 +120879.157}
SPL {X  -155.811, Y  +731.738, Z    +0.000, E1   -70.890, E3 +120888.165}
SPL {X  -152.643, Y  +739.844, Z    +0.000, E1   -70.463, E3 +120897.024}
SPL {X  -149.782, Y  +746.247, Z    +0.000, E1   -70.149, E3 +120903.714}
SPL {X  -146.450, Y  +752.910, Z    +0.000, E1   -69.680, E3 +120911.592}
SPL {X  -143.017, Y  +759.082, Z    +0.000, E1   -69.156, E3 +120919.204}
SPL {X  -140.057, Y  +763.953, Z    +0.000, E1   -68.829, E3 +120924.443}
SPL {X  -136.535, Y  +769.298, Z    +0.000, E1   -68.442, E3 +120930.305}
SPL {X  -133.553, Y  +773.498, Z    +0.000, E1   -67.773, E3 +120936.470}
SPL {X  -129.830, Y  +778.379, Z    +0.000, E1   -67.491, E3 +120941.095}
SPL {X  -116.788, Y  +792.975, Z    +0.000, E1   -71.297, E3 +120934.480}
SPL {X   -64.927, Y  +827.895, Z    +0.000, E1   -57.691, E3 +121060.083}
ENDSPLINE

SPLINE
SPL {X  -111.648, Y  +797.871, Z    +0.000, E1   -60.847, E3 +121257.065}
SPL {X  -149.288, Y  +747.285, Z    +0.000, E1   -46.770, E3 +121253.056}
SPL {X  -159.627, Y  +719.761, Z    +0.000, E1   -35.247, E3 +121258.121}
SPL {X  -164.185, Y  +697.485, Z    +0.000, E1   -20.950, E3 +121258.440}
SPL {X  -165.594, Y  +679.817, Z    +0.000, E1    -6.204, E3 +121257.216}
SPL {X  -165.650, Y  +673.522, Z    +0.000, E1    -0.038, E3 +121256.185}
SPL {X  -165.650, Y  +671.354, Z    +0.000, E1    +3.728, E3 +121255.673}
SPL {X  -165.650, Y  +666.485, Z    +0.000, E1   +14.169, E3 +121255.400}
SPL {X  -165.650, Y  +661.236, Z    +0.000, E1   +26.072, E3 +121255.089}
SPL {X  -165.650, Y  +655.357, Z    +0.000, E1   +38.693, E3 +121254.317}
SPL {X  -165.650, Y  +646.637, Z    +0.000, E1   +52.169, E3 +121254.098}
SPL {X  -165.650, Y  +637.909, Z    +0.000, E1   +64.161, E3 +121250.894}
SPL {X  -165.650, Y  +618.963, Z    +0.000, E1   +72.815, E3 +121251.957}
SPL {X  -165.650, Y  +575.208, Z    +0.000, E1   +76.222, E3 +121263.218}
SPL {X  -165.650, Y  +394.754, Z    +0.000, E1   +73.248, E3 +121358.364}
ENDSPLINE

SPLINE
SPL {X  -165.650, Y  +407.500, Z    +0.000, E1   +70.919, E3 +121372.985}
ENDSPLINE

SPLINE
SPL {X  -165.650, Y  +390.855, Z    +0.000, E1   +71.004, E3 +121383.913}
SPL {X  -165.534, Y  +372.295, Z    +0.000, E1   +71.066, E3 +121396.463}
SPL {X  -164.039, Y  +355.451, Z    +0.000, E1   +70.703, E3 +121411.862}
SPL {X  -161.297, Y  +340.777, Z    +0.000, E1   +70.794, E3 +121421.154}
ENDSPLINE

SPLINE
SPL {X  -162.352, Y  +345.609, Z    +0.000, E1   +69.290, E3 +121431.087}
ENDSPLINE

SPLINE
SPL {X  -159.253, Y  +332.909, Z    +0.000, E1   +69.652, E3 +121437.434}
SPL {X  -155.267, Y  +320.775, Z    +0.000, E1   +69.854, E3 +121444.527}
SPL {X  -151.256, Y  +310.961, Z    +0.000, E1   +69.467, E3 +121454.402}
SPL {X  -148.628, Y  +305.359, Z    +0.000, E1   +68.848, E3 +121462.680}
SPL {X  -145.495, Y  +299.310, Z    +0.000, E1   +68.659, E3 +121468.240}
SPL {X  -142.111, Y  +293.387, Z    +0.000, E1   +68.421, E3 +121473.881}
SPL {X  -138.525, Y  +287.667, Z    +0.000, E1   +67.662, E3 +121482.441}
SPL {X  -134.450, Y  +281.737, Z    +0.000, E1   +67.268, E3 +121488.546}
SPL {X  -131.812, Y  +278.173, Z    +0.000, E1   +66.669, E3 +121493.895}
SPL {X  -128.148, Y  +273.533, Z    +0.000, E1   +67.328, E3 +121494.253}
SPL {X  -116.216, Y  +260.459, Z    +0.000, E1   +70.200, E3 +121490.560}
SPL {X   -66.125, Y  +226.621, Z    +0.000, E1   +55.862, E3 +121653.458}
ENDSPLINE

SPLINE
SPL {X  -111.531, Y  +256.023, Z    +0.000, E1   +58.853, E3 +121796.340}
SPL {X  -139.240, Y  +288.767, Z    +0.000, E1   +52.898, E3 +121806.513}
SPL {X  -156.827, Y  +325.161, Z    +0.000, E1   +39.042, E3 +121804.882}
SPL {X  -163.133, Y  +349.734, Z    +0.000, E1   +25.193, E3 +121806.007}
SPL {X  -165.214, Y  +366.494, Z    +0.000, E1   +12.605, E3 +121805.480}
SPL {X  -165.615, Y  +375.073, Z    +0.000, E1    +5.133, E3 +121804.967}
SPL {X  -165.650, Y  +380.392, Z    +0.000, E1    +0.180, E3 +121803.926}
SPL {X  -165.650, Y  +381.828, Z    +0.000, E1    -2.219, E3 +121803.324}
SPL {X  -165.650, Y  +385.044, Z    +0.000, E1    -8.496, E3 +121803.124}
SPL {X  -165.650, Y  +388.717, Z    +0.000, E1   -16.400, E3 +121802.980}
SPL {X  -165.650, Y  +394.613, Z    +0.000, E1   -29.184, E3 +121802.448}
SPL {X  -165.650, Y  +402.836, Z    +0.000, E1   -44.797, E3 +121801.851}
SPL {X  -165.650, Y  +416.111, Z    +0.000, E1   -60.729, E3 +121800.917}
SPL {X  -165.650, Y  +471.994, Z    +0.000, E1   -75.670, E3 +121808.971}
SPL {X  -164.204, Y  +697.342, Z    +0.000, E1   -76.015, E3 +121896.994}
ENDSPLINE

SPLINE
SPL {X  -165.650, Y  +664.340, Z    +0.000, E1   -71.862, E3 +121922.397}
ENDSPLINE

SPLINE
SPL {X  -165.237, Y  +687.187, Z    +0.000, E1   -71.947, E3 +121936.659}
SPL {X  -163.865, Y  +699.752, Z    +0.000, E1   -71.643, E3 +121948.064}
SPL {X  -161.821, Y  +710.908, Z    +0.000, E1   -71.322, E3 +121958.604}
SPL {X  -158.993, Y  +721.987, Z    +0.000, E1   -71.173, E3 +121967.393}
SPL {X  -155.811, Y  +731.738, Z    +0.000, E1   -70.890, E3 +121976.401}
SPL {X  -152.643, Y  +739.844, Z    +0.000, E1   -70.463, E3 +121985.260}
SPL {X  -149.782, Y  +746.247, Z    +0.000, E1   -70.149, E3 +121991.950}
SPL {X  -146.450, Y  +752.910, Z    +0.000, E1   -69.680, E3 +121999.828}
SPL {X  -143.017, Y  +759.082, Z    +0.000, E1   -69.156, E3 +122007.439}
SPL {X  -139.030, Y  +765.558, Z    +0.000, E1   -68.719, E3 +122014.472}
SPL {X  -134.589, Y  +772.070, Z    +0.000, E1   -68.090, E3 +122022.321}
SPL {X  -129.830, Y  +778.379, Z    +0.000, E1   -67.491, E3 +122029.331}
SPL {X  -116.788, Y  +792.975, Z    +0.000, E1   -71.297, E3 +122022.715}
SPL {X   -64.927, Y  +827.895, Z    +0.000, E1   -57.691, E3 +122148.318}
ENDSPLINE

SPLINE
SPL {X  -111.648, Y  +797.871, Z    +0.000, E1   -60.847, E3 +122345.300}
SPL {X  -149.288, Y  +747.285, Z    +0.000, E1   -46.770, E3 +122341.291}
SPL {X  -159.627, Y  +719.761, Z    +0.000, E1   -35.247, E3 +122346.356}
SPL {X  -164.185, Y  +697.485, Z    +0.000, E1   -20.950, E3 +122346.675}
SPL {X  -165.594, Y  +679.817, Z    +0.000, E1    -6.204, E3 +122345.451}
SPL {X  -165.650, Y  +673.522, Z    +0.000, E1    -0.038, E3 +122344.420}
SPL {X  -165.650, Y  +671.354, Z    +0.000, E1    +3.728, E3 +122343.908}
SPL {X  -165.650, Y  +666.485, Z    +0.000, E1   +14.169, E3 +122343.635}
SPL {X  -165.650, Y  +661.236, Z    +0.000, E1   +26.072, E3 +122343.324}
SPL {X  -165.650, Y  +653.063, Z    +0.000, E1   +42.395, E3 +122342.728}
SPL {X  -165.650, Y  +640.535, Z    +0.000, E1   +60.776, E3 +122340.213}
SPL {X  -165.650, Y  +618.963, Z    +0.000, E1   +72.815, E3 +122340.192}
SPL {X  -165.650, Y  +582.897, Z    +0.000, E1   +76.147, E3 +122348.854}
SPL {X  -165.650, Y  +558.388, Z    +0.000, E1   +76.294, E3 +122357.166}
SPL {X  -165.650, Y  +391.690, Z    +0.000, E1   +75.504, E3 +122426.932}
ENDSPLINE

SPLINE
SPL {X  -165.650, Y  +396.283, Z    +0.000, E1   +72.775, E3 +122450.237}
SPL {X  -165.650, Y  +407.500, Z    +0.000, E1   +70.919, E3 +122461.221}
ENDSPLINE

SPLINE
SPL {X  -165.650, Y  +384.687, Z    +0.000, E1   +71.028, E3 +122476.466}
SPL {X  -164.996, Y  +363.797, Z    +0.000, E1   +70.987, E3 +122491.442}
SPL {X  -162.841, Y  +348.123, Z    +0.000, E1   +70.683, E3 +122505.369}
SPL {X  -162.352, Y  +345.609, Z    +0.000, E1   +69.290, E3 +122519.322}
SPL {X  -157.663, Y  +327.685, Z    +0.000, E1   +69.808, E3 +122528.183}
SPL {X  -152.892, Y  +314.750, Z    +0.000, E1   +69.675, E3 +122538.398}
SPL {X  -149.246, Y  +306.628, Z    +0.000, E1   +69.029, E3 +122548.866}
SPL {X  -144.614, Y  +297.712, Z    +0.000, E1   +68.717, E3 +122557.220}
SPL {X  -141.011, Y  +291.576, Z    +0.000, E1   +68.040, E3 +122565.698}
SPL {X  -137.649, Y  +286.345, Z    +0.000, E1   +67.498, E3 +122572.391}
SPL {X  -134.450, Y  +281.737, Z    +0.000, E1   +67.268, E3 +122576.782}
SPL {X  -131.812, Y  +278.173, Z    +0.000, E1   +66.669, E3 +122582.130}
SPL {X  -128.148, Y  +273.533, Z    +0.000, E1   +67.328, E3 +122582.489}
SPL {X  -116.216, Y  +260.459, Z    +0.000, E1   +70.200, E3 +122578.795}
SPL {X   -66.125, Y  +226.621, Z    +0.000, E1   +55.862, E3 +122741.693}
ENDSPLINE

SPLINE
SPL {X  -111.531, Y  +256.023, Z    +0.000, E1   +58.853, E3 +122884.575}
SPL {X  -139.240, Y  +288.767, Z    +0.000, E1   +52.898, E3 +122894.748}
SPL {X  -156.827, Y  +325.161, Z    +0.000, E1   +39.042, E3 +122893.117}
SPL {X  -162.324, Y  +345.471, Z    +0.000, E1   +27.849, E3 +122893.586}
SPL {X  -165.055, Y  +364.477, Z    +0.000, E1   +14.326, E3 +122894.024}
SPL {X  -165.646, Y  +377.353, Z    +0.000, E1    +3.112, E3 +122892.981}
SPL {X  -165.650, Y  +380.500, Z    +0.000, E1    -0.000, E3 +122892.107}
SPL {X  -165.650, Y  +381.828, Z    +0.000, E1    -2.219, E3 +122891.559}
SPL {X  -165.650, Y  +385.044, Z    +0.000, E1    -8.496, E3 +122891.359}
SPL {X  -165.650, Y  +388.717, Z    +0.000, E1   -16.400, E3 +122891.215}
SPL {X  -165.650, Y  +394.613, Z    +0.000, E1   -29.184, E3 +122890.684}
SPL {X  -165.650, Y  +402.836, Z    +0.000, E1   -44.797, E3 +122890.086}
SPL {X  -165.650, Y  +416.111, Z    +0.000, E1   -60.729, E3 +122889.153}
SPL {X  -165.650, Y  +471.994, Z    +0.000, E1   -75.670, E3 +122897.206}
SPL {X  -164.204, Y  +697.342, Z    +0.000, E1   -76.015, E3 +122985.229}
ENDSPLINE

SPLINE
SPL {X  -165.650, Y  +656.030, Z    +0.000, E1   -71.686, E3 +123006.668}
ENDSPLINE

SPLINE
SPL {X  -165.610, Y  +679.119, Z    +0.000, E1   -71.889, E3 +123020.292}
SPL {X  -164.561, Y  +694.465, Z    +0.000, E1   -71.736, E3 +123031.925}
SPL {X  -162.089, Y  +709.665, Z    +0.000, E1   -71.739, E3 +123042.126}
SPL {X  -159.776, Y  +719.221, Z    +0.000, E1   -71.038, E3 +123054.948}
SPL {X  -155.811, Y  +731.738, Z    +0.000, E1   -70.890, E3 +123064.636}
SPL {X  -152.643, Y  +739.844, Z    +0.000, E1   -70.463, E3 +123073.495}
SPL {X  -149.782, Y  +746.247, Z    +0.000, E1   -70.149, E3 +123080.185}
SPL {X  -146.450, Y  +752.910, Z    +0.000, E1   -69.680, E3 +123088.063}
SPL {X  -143.017, Y  +759.082, Z    +0.000, E1   -69.156, E3 +123095.674}
SPL {X  -139.030, Y  +765.558, Z    +0.000, E1   -68.719, E3 +123102.707}
SPL {X  -135.682, Y  +770.527, Z    +0.000, E1   -68.337, E3 +123108.091}
SPL {X  -132.359, Y  +775.105, Z    +0.000, E1   -67.661, E3 +123114.633}
SPL {X  -128.720, Y  +779.765, Z    +0.000, E1   -67.454, E3 +123118.614}
SPL {X  -116.788, Y  +792.975, Z    +0.000, E1   -71.297, E3 +123110.950}
SPL {X   -64.927, Y  +827.895, Z    +0.000, E1   -57.691, E3 +123236.553}
ENDSPLINE

SPLINE
SPL {X  -111.648, Y  +797.871, Z    +0.000, E1   -60.847, E3 +123433.536}
SPL {X  -149.288, Y  +747.285, Z    +0.000, E1   -46.770, E3 +123429.526}
SPL {X  -159.627, Y  +719.761, Z    +0.000, E1   -35.247, E3 +123434.591}
SPL {X  -164.185, Y  +697.485, Z    +0.000, E1   -20.950, E3 +123434.910}
SPL {X  -165.594, Y  +679.817, Z    +0.000, E1    -6.204, E3 +123433.687}
SPL {X  -165.650, Y  +673.522, Z    +0.000, E1    -0.038, E3 +123432.656}
SPL {X  -165.650, Y  +671.354, Z    +0.000, E1    +3.728, E3 +123432.143}
SPL {X  -165.650, Y  +666.485, Z    +0.000, E1   +14.169, E3 +123431.870}
SPL {X  -165.650, Y  +661.236, Z    +0.000, E1   +26.072, E3 +123431.560}
SPL {X  -165.650, Y  +653.063, Z    +0.000, E1   +42.395, E3 +123430.964}
SPL {X  -165.650, Y  +640.535, Z    +0.000, E1   +60.776, E3 +123428.449}
SPL {X  -165.650, Y  +618.963, Z    +0.000, E1   +72.815, E3 +123428.428}
SPL {X  -165.650, Y  +575.208, Z    +0.000, E1   +76.222, E3 +123439.688}
SPL {X  -165.650, Y  +394.754, Z    +0.000, E1   +73.248, E3 +123534.835}
ENDSPLINE

SPLINE
SPL {X  -165.650, Y  +407.500, Z    +0.000, E1   +70.919, E3 +123549.456}
ENDSPLINE

SPLINE
SPL {X  -165.650, Y  +390.855, Z    +0.000, E1   +71.004, E3 +123560.384}
SPL {X  -165.534, Y  +372.295, Z    +0.000, E1   +71.066, E3 +123572.934}
SPL {X  -164.039, Y  +355.451, Z    +0.000, E1   +70.703, E3 +123588.332}
SPL {X  -161.297, Y  +340.777, Z    +0.000, E1   +70.794, E3 +123597.624}
ENDSPLINE

SPLINE
SPL {X  -162.352, Y  +345.609, Z    +0.000, E1   +69.290, E3 +123607.558}
ENDSPLINE

SPLINE
SPL {X  -157.663, Y  +327.685, Z    +0.000, E1   +69.808, E3 +123616.418}
SPL {X  -152.892, Y  +314.750, Z    +0.000, E1   +69.675, E3 +123626.634}
SPL {X  -149.246, Y  +306.628, Z    +0.000, E1   +69.029, E3 +123637.102}
SPL {X  -145.495, Y  +299.310, Z    +0.000, E1   +68.659, E3 +123644.710}
SPL {X  -142.111, Y  +293.387, Z    +0.000, E1   +68.421, E3 +123650.352}
SPL {X  -138.525, Y  +287.667, Z    +0.000, E1   +67.662, E3 +123658.912}
SPL {X  -134.450, Y  +281.737, Z    +0.000, E1   +67.268, E3 +123665.017}
SPL {X  -131.812, Y  +278.173, Z    +0.000, E1   +66.669, E3 +123670.365}
SPL {X  -128.148, Y  +273.533, Z    +0.000, E1   +67.328, E3 +123670.724}
SPL {X  -116.216, Y  +260.459, Z    +0.000, E1   +70.200, E3 +123667.030}
SPL {X   -66.125, Y  +226.621, Z    +0.000, E1   +55.862, E3 +123829.929}
ENDSPLINE

SPLINE
SPL {X  -111.531, Y  +256.023, Z    +0.000, E1   +58.853, E3 +123972.810}
SPL {X  -139.240, Y  +288.767, Z    +0.000, E1   +52.898, E3 +123982.983}
SPL {X  -156.827, Y  +325.161, Z    +0.000, E1   +39.042, E3 +123981.353}
SPL {X  -162.324, Y  +345.471, Z    +0.000, E1   +27.849, E3 +123981.821}
SPL {X  -165.055, Y  +364.477, Z    +0.000, E1   +14.326, E3 +123982.260}
SPL {X  -165.646, Y  +377.353, Z    +0.000, E1    +3.112, E3 +123981.216}
SPL {X  -165.650, Y  +380.500, Z    +0.000, E1    -0.000, E3 +123980.342}
SPL {X  -165.650, Y  +381.828, Z    +0.000, E1    -2.219, E3 +123979.795}
SPL {X  -165.650, Y  +385.044, Z    +0.000, E1    -8.496, E3 +123979.594}
SPL {X  -165.650, Y  +390.492, Z    +0.000, E1   -20.084, E3 +123979.249}
SPL {X  -165.650, Y  +400.081, Z    +0.000, E1   -39.836, E3 +123978.554}
SPL {X  -165.650, Y  +416.111, Z    +0.000, E1   -60.729, E3 +123977.388}
SPL {X  -165.650, Y  +471.994, Z    +0.000, E1   -75.670, E3 +123985.441}
SPL {X  -164.204, Y  +697.342, Z    +0.000, E1   -76.015, E3 +124073.464}
ENDSPLINE

SPLINE
SPL {X  -165.650, Y  +656.030, Z    +0.000, E1   -71.686, E3 +124094.904}
ENDSPLINE

SPLINE
SPL {X  -165.472, Y  +683.167, Z    +0.000, E1   -72.022, E3 +124109.912}
SPL {X  -163.865, Y  +699.752, Z    +0.000, E1   -71.643, E3 +124124.535}
SPL {X  -161.571, Y  +712.032, Z    +0.000, E1   -71.595, E3 +124133.128}
SPL {X  -159.776, Y  +719.221, Z    +0.000, E1   -71.038, E3 +124143.183}
SPL {X  -155.811, Y  +731.738, Z    +0.000, E1   -70.890, E3 +124152.871}
SPL {X  -152.643, Y  +739.844, Z    +0.000, E1   -70.463, E3 +124161.730}
SPL {X  -149.782, Y  +746.247, Z    +0.000, E1   -70.149, E3 +124168.420}
SPL {X  -146.450, Y  +752.910, Z    +0.000, E1   -69.680, E3 +124176.298}
SPL {X  -143.017, Y  +759.082, Z    +0.000, E1   -69.156, E3 +124183.909}
SPL {X  -140.057, Y  +763.953, Z    +0.000, E1   -68.829, E3 +124189.149}
SPL {X  -136.535, Y  +769.298, Z    +0.000, E1   -68.442, E3 +124195.011}
SPL {X  -133.553, Y  +773.498, Z    +0.000, E1   -67.773, E3 +124201.175}
SPL {X  -129.830, Y  +778.379, Z    +0.000, E1   -67.491, E3 +124205.801}
SPL {X  -116.788, Y  +792.975, Z    +0.000, E1   -71.297, E3 +124199.185}
SPL {X   -70.520, Y  +825.390, Z    +0.000, E1   -59.928, E3 +124293.096}
SPL {X   -62.607, Y  +828.863, Z    +0.000, E1   -56.584, E3 +124347.980}
ENDSPLINE

SPLINE
SPL {X  -111.648, Y  +797.871, Z    +0.000, E1   -60.847, E3 +124521.771}
SPL {X  -149.288, Y  +747.285, Z    +0.000, E1   -46.770, E3 +124517.762}
SPL {X  -161.496, Y  +712.364, Z    +0.000, E1   -31.137, E3 +124523.557}
SPL {X  -164.701, Y  +693.202, Z    +0.000, E1   -17.512, E3 +124522.531}
SPL {X  -165.453, Y  +683.578, Z    +0.000, E1    -9.445, E3 +124521.733}
SPL {X  -165.642, Y  +677.105, Z    +0.000, E1    -3.559, E3 +124522.043}
SPL {X  -165.650, Y  +673.522, Z    +0.000, E1    -0.038, E3 +124520.891}
SPL {X  -165.650, Y  +671.354, Z    +0.000, E1    +3.728, E3 +124520.379}
SPL {X  -165.650, Y  +666.485, Z    +0.000, E1   +14.169, E3 +124520.106}
SPL {X  -165.650, Y  +661.236, Z    +0.000, E1   +26.072, E3 +124519.795}
SPL {X  -165.650, Y  +655.357, Z    +0.000, E1   +38.693, E3 +124519.023}
SPL {X  -165.650, Y  +646.637, Z    +0.000, E1   +52.169, E3 +124518.804}
SPL {X  -165.650, Y  +637.909, Z    +0.000, E1   +64.161, E3 +124515.600}
SPL {X  -165.650, Y  +618.963, Z    +0.000, E1   +72.815, E3 +124516.663}
SPL {X  -165.650, Y  +575.208, Z    +0.000, E1   +76.222, E3 +124527.924}
SPL {X  -165.650, Y  +394.754, Z    +0.000, E1   +73.248, E3 +124623.070}
ENDSPLINE

SPLINE
SPL {X  -165.650, Y  +407.500, Z    +0.000, E1   +70.919, E3 +124637.691}
ENDSPLINE

SPLINE
SPL {X  -165.650, Y  +390.855, Z    +0.000, E1   +71.004, E3 +124648.619}
SPL {X  -165.534, Y  +372.295, Z    +0.000, E1   +71.066, E3 +124661.169}
SPL {X  -164.039, Y  +355.451, Z    +0.000, E1   +70.703, E3 +124676.567}
SPL {X  -161.297, Y  +340.777, Z    +0.000, E1   +70.794, E3 +124685.860}
ENDSPLINE

SPLINE
SPL {X  -162.352, Y  +345.609, Z    +0.000, E1   +69.290, E3 +124695.793}
ENDSPLINE

SPLINE
SPL {X  -157.663, Y  +327.685, Z    +0.000, E1   +69.808, E3 +124704.653}
SPL {X  -152.892, Y  +314.750, Z    +0.000, E1   +69.675, E3 +124714.869}
SPL {X  -149.246, Y  +306.628, Z    +0.000, E1   +69.029, E3 +124725.337}
SPL {X  -144.614, Y  +297.712, Z    +0.000, E1   +68.717, E3 +124733.691}
SPL {X  -141.011, Y  +291.576, Z    +0.000, E1   +68.040, E3 +124742.169}
SPL {X  -137.649, Y  +286.345, Z    +0.000, E1   +67.498, E3 +124748.862}
SPL {X  -134.450, Y  +281.737, Z    +0.000, E1   +67.268, E3 +124753.252}
SPL {X  -131.812, Y  +278.173, Z    +0.000, E1   +66.669, E3 +124758.601}
SPL {X  -128.148, Y  +273.533, Z    +0.000, E1   +67.328, E3 +124758.959}
SPL {X  -116.216, Y  +260.459, Z    +0.000, E1   +70.200, E3 +124755.266}
SPL {X   -66.125, Y  +226.621, Z    +0.000, E1   +55.862, E3 +124918.164}
ENDSPLINE

SPLINE
SPL {X  -111.531, Y  +256.023, Z    +0.000, E1   +58.853, E3 +125061.046}
SPL {X  -139.240, Y  +288.767, Z    +0.000, E1   +52.898, E3 +125071.219}
SPL {X  -156.827, Y  +325.161, Z    +0.000, E1   +39.042, E3 +125069.588}
SPL {X  -162.324, Y  +345.471, Z    +0.000, E1   +27.849, E3 +125070.057}
SPL {X  -165.055, Y  +364.477, Z    +0.000, E1   +14.326, E3 +125070.495}
SPL {X  -165.646, Y  +377.353, Z    +0.000, E1    +3.112, E3 +125069.452}
SPL {X  -165.650, Y  +380.500, Z    +0.000, E1    -0.000, E3 +125068.578}
SPL {X  -165.650, Y  +381.828, Z    +0.000, E1    -2.219, E3 +125068.030}
SPL {X  -165.650, Y  +385.044, Z    +0.000, E1    -8.496, E3 +125067.830}
SPL {X  -165.650, Y  +388.717, Z    +0.000, E1   -16.400, E3 +125067.685}
SPL {X  -165.650, Y  +394.613, Z    +0.000, E1   -29.184, E3 +125067.154}
SPL {X  -165.650, Y  +402.836, Z    +0.000, E1   -44.797, E3 +125066.557}
SPL {X  -165.650, Y  +416.111, Z    +0.000, E1   -60.729, E3 +125065.623}
SPL {X  -165.650, Y  +471.994, Z    +0.000, E1   -75.670, E3 +125073.677}
SPL {X  -164.204, Y  +697.342, Z    +0.000, E1   -76.015, E3 +125161.699}
ENDSPLINE

SPLINE
SPL {X  -165.650, Y  +656.030, Z    +0.000, E1   -71.686, E3 +125183.139}
ENDSPLINE

SPLINE
SPL {X  -165.610, Y  +679.119, Z    +0.000, E1   -71.889, E3 +125196.762}
SPL {X  -164.561, Y  +694.465, Z    +0.000, E1   -71.736, E3 +125208.395}
SPL {X  -162.089, Y  +709.665, Z    +0.000, E1   -71.739, E3 +125218.596}
SPL {X  -159.776, Y  +719.221, Z    +0.000, E1   -71.038, E3 +125231.418}
SPL {X  -155.811, Y  +731.738, Z    +0.000, E1   -70.890, E3 +125241.106}
SPL {X  -152.643, Y  +739.844, Z    +0.000, E1   -70.463, E3 +125249.966}
SPL {X  -149.782, Y  +746.247, Z    +0.000, E1   -70.149, E3 +125256.655}
SPL {X  -146.450, Y  +752.910, Z    +0.000, E1   -69.680, E3 +125264.534}
SPL {X  -143.017, Y  +759.082, Z    +0.000, E1   -69.156, E3 +125272.145}
SPL {X  -140.057, Y  +763.953, Z    +0.000, E1   -68.829, E3 +125277.384}
SPL {X  -136.535, Y  +769.298, Z    +0.000, E1   -68.442, E3 +125283.246}
SPL {X  -133.553, Y  +773.498, Z    +0.000, E1   -67.773, E3 +125289.411}
SPL {X  -129.830, Y  +778.379, Z    +0.000, E1   -67.491, E3 +125294.037}
SPL {X  -116.788, Y  +792.975, Z    +0.000, E1   -71.297, E3 +125287.421}
SPL {X   -64.927, Y  +827.895, Z    +0.000, E1   -57.691, E3 +125413.024}
ENDSPLINE

SPLINE
SPL {X  -111.648, Y  +797.871, Z    +0.000, E1   -60.847, E3 +125610.006}
SPL {X  -149.288, Y  +747.285, Z    +0.000, E1   -46.770, E3 +125605.997}
SPL {X  -159.627, Y  +719.761, Z    +0.000, E1   -35.247, E3 +125611.062}
SPL {X  -164.185, Y  +697.485, Z    +0.000, E1   -20.950, E3 +125611.381}
SPL {X  -165.594, Y  +679.817, Z    +0.000, E1    -6.204, E3 +125610.157}
SPL {X  -165.650, Y  +673.522, Z    +0.000, E1    -0.038, E3 +125609.126}
SPL {X  -165.650, Y  +671.354, Z    +0.000, E1    +3.728, E3 +125608.614}
SPL {X  -165.650, Y  +666.485, Z    +0.000, E1   +14.169, E3 +125608.341}
SPL {X  -165.650, Y  +661.236, Z    +0.000, E1   +26.072, E3 +125608.030}
SPL {X  -165.650, Y  +653.063, Z    +0.000, E1   +42.395, E3 +125607.434}
SPL {X  -165.650, Y  +640.535, Z    +0.000, E1   +60.776, E3 +125604.919}
SPL {X  -165.650, Y  +618.963, Z    +0.000, E1   +72.815, E3 +125604.898}
SPL {X  -165.650, Y  +575.208, Z    +0.000, E1   +76.222, E3 +125616.159}
SPL {X  -165.650, Y  +394.754, Z    +0.000, E1   +73.248, E3 +125711.305}
ENDSPLINE

SPLINE
SPL {X  -165.650, Y  +407.500, Z    +0.000, E1   +70.919, E3 +125725.927}
ENDSPLINE

SPLINE
SPL {X  -165.650, Y  +390.855, Z    +0.000, E1   +71.004, E3 +125736.854}
SPL {X  -165.534, Y  +372.295, Z    +0.000, E1   +71.066, E3 +125749.405}
SPL {X  -164.687, Y  +360.663, Z    +0.000, E1   +70.826, E3 +125759.696}
SPL {X  -162.841, Y  +348.123, Z    +0.000, E1   +70.683, E3 +125770.075}
SPL {X  -162.352, Y  +345.609, Z    +0.000, E1   +69.290, E3 +125784.028}
SPL {X  -157.663, Y  +327.685, Z    +0.000, E1   +69.808, E3 +125792.889}
SPL {X  -154.072, Y  +317.659, Z    +0.000, E1   +69.748, E3 +125800.380}
SPL {X  -151.256, Y  +310.961, Z    +0.000, E1   +69.467, E3 +125807.343}
SPL {X  -148.628, Y  +305.359, Z    +0.000, E1   +68.848, E3 +125815.622}
SPL {X  -145.495, Y  +299.310, Z    +0.000, E1   +68.659, E3 +125821.181}
SPL {X  -142.111, Y  +293.387, Z    +0.000, E1   +68.421, E3 +125826.823}
SPL {X  -138.525, Y  +287.667, Z    +0.000, E1   +67.662, E3 +125835.382}
SPL {X  -134.450, Y  +281.737, Z    +0.000, E1   +67.268, E3 +125841.488}
SPL {X  -131.812, Y  +278.173, Z    +0.000, E1   +66.669, E3 +125846.836}
SPL {X  -128.148, Y  +273.533, Z    +0.000, E1   +67.328, E3 +125847.194}
SPL {X  -116.216, Y  +260.459, Z    +0.000, E1   +70.200, E3 +125843.501}
SPL {X   -67.926, Y  +227.417, Z    +0.000, E1   +56.698, E3 +125978.220}
SPL {X   -66.052, Y  +226.589, Z    +0.000, E1   +55.637, E3 +126031.453}
ENDSPLINE

SPLINE
SPL {X  -111.531, Y  +256.023, Z    +0.000, E1   +58.853, E3 +126149.281}
SPL {X  -139.240, Y  +288.767, Z    +0.000, E1   +52.898, E3 +126159.454}
SPL {X  -156.827, Y  +325.161, Z    +0.000, E1   +39.042, E3 +126157.823}
SPL {X  -162.324, Y  +345.471, Z    +0.000, E1   +27.849, E3 +126158.292}
SPL {X  -164.696, Y  +360.744, Z    +0.000, E1   +17.229, E3 +126159.206}
SPL {X  -165.561, Y  +373.081, Z    +0.000, E1    +6.973, E3 +126157.950}
SPL {X  -165.650, Y  +380.800, Z    +0.000, E1    -0.199, E3 +126156.696}
SPL {X  -165.650, Y  +385.044, Z    +0.000, E1    -8.496, E3 +126156.065}
SPL {X  -165.650, Y  +390.492, Z    +0.000, E1   -20.084, E3 +126155.719}
SPL {X  -165.650, Y  +398.793, Z    +0.000, E1   -37.509, E3 +126155.237}
SPL {X  -165.650, Y  +409.325, Z    +0.000, E1   -54.181, E3 +126153.917}
SPL {X  -165.650, Y  +420.423, Z    +0.000, E1   -63.808, E3 +126154.066}
SPL {X  -165.650, Y  +471.994, Z    +0.000, E1   -75.670, E3 +126161.912}
SPL {X  -164.204, Y  +697.342, Z    +0.000, E1   -76.015, E3 +126249.935}
ENDSPLINE

SPLINE
SPL {X  -165.650, Y  +656.030, Z    +0.000, E1   -71.686, E3 +126271.374}
ENDSPLINE

SPLINE
SPL {X  -165.610, Y  +679.119, Z    +0.000, E1   -71.889, E3 +126284.997}
SPL {X  -163.827, Y  +700.009, Z    +0.000, E1   -71.824, E3 +126299.563}
SPL {X  -161.821, Y  +710.908, Z    +0.000, E1   -71.322, E3 +126311.545}
SPL {X  -158.993, Y  +721.987, Z    +0.000, E1   -71.173, E3 +126320.334}
SPL {X  -155.811, Y  +731.738, Z    +0.000, E1   -70.890, E3 +126329.342}
SPL {X  -152.643, Y  +739.844, Z    +0.000, E1   -70.463, E3 +126338.201}
SPL {X  -149.782, Y  +746.247, Z    +0.000, E1   -70.149, E3 +126344.891}
SPL {X  -146.450, Y  +752.910, Z    +0.000, E1   -69.680, E3 +126352.769}
SPL {X  -143.017, Y  +759.082, Z    +0.000, E1   -69.156, E3 +126360.380}
SPL {X  -139.030, Y  +765.558, Z    +0.000, E1   -68.719, E3 +126367.413}
SPL {X  -135.682, Y  +770.527, Z    +0.000, E1   -68.337, E3 +126372.797}
SPL {X  -132.359, Y  +775.105, Z    +0.000, E1   -67.661, E3 +126379.338}
SPL {X  -128.720, Y  +779.765, Z    +0.000, E1   -67.454, E3 +126383.319}
SPL {X  -116.788, Y  +792.975, Z    +0.000, E1   -71.297, E3 +126375.656}
SPL {X   -64.927, Y  +827.895, Z    +0.000, E1   -57.691, E3 +126501.259}
ENDSPLINE

